(* Logix 5000 project; controller Almacen_2 vendor 1 type 14 code 235 rev 36.11; software revision 36.00 *)

TASK MainTask (continuous, watchdog 500 ms) : MainProgram
TASK SafetyTask (periodic, rate 20 ms, priority 10, watchdog 20 ms) : SafetyProgram

MODULES
   Local : vendor 1 type 14 code 235 (5069 0, rev 36.11)
      EN2TR_Principal : vendor 1 type 12 code 200 (Ethernet 10.12.143.10, rev 10.7, Output RPI 10 ms)
           Point_IO_Conveyor_2:10:O.0   // Spare
           Point_IO_Conveyor_2:10:O.1   // Spare
           Point_IO_Conveyor_2:10:O.2   // Spare
           Point_IO_Conveyor_2:10:O.3   // Spare
           Point_IO_Conveyor_2:10:O.4   // Spare
           Point_IO_Conveyor_2:10:O.5   // Spare
           Point_IO_Conveyor_2:10:O.6   // Spare
           Point_IO_Conveyor_2:10:O.7   // Spare
           Point_IO_Conveyor_2:8:O.5   // Spare
           Point_IO_Conveyor_2:8:O.0   // Reset Válvula General Conveyor 2
           Point_IO_Conveyor_2:8:O.1   // Señal de Impresion de Marcadora Laser
           Point_IO_Conveyor_2:8:O.2   // Lampara indicadora izquierda
           Point_IO_Conveyor_2:8:O.3   // Lampara Cognex 2
           Point_IO_Conveyor_2:8:O.4   // Lampara Cognex 1
           Point_IO_Conveyor_2:8:O.6   // Spare
           Point_IO_Conveyor_2:8:O.7   // Spare
           Point_IO_Almacen_2:1:I.2   // Sensor Piston 1 Horizontal Izquierda
           Point_IO_Almacen_2:1:I.3   // Sensor Piston 1 Horizontal Derecha
           Point_IO_Almacen_2:1:I.4   // Disponible
           Point_IO_Almacen_2:1:I.5   // Sensor Piston 2 Vertical Atras
           Point_IO_Almacen_2:1:I.6   // Sensor Piston 4 Giro Direccion Conveyor
           Point_IO_Almacen_2:1:I.7   // Sensor Piston 4 Giro Direccion Almacen
           Point_IO_Almacen_2:1:I.0   // Disponible
           Point_IO_Almacen_2:1:I.1   // Sensor Piston 3 Griper Arriba
           Point_IO_Conveyor_2:5:I.0   // Sensor Limit Switch Tope
           Point_IO_Conveyor_2:5:I.1   // Sensor Inductivo Entrada desde Almacén (Inicial)
           Point_IO_Conveyor_2:5:I.2   // Robot Fanuc Fence Open
           Point_IO_Conveyor_2:5:I.3   // Robot Fanuc E Stop
           Point_IO_Conveyor_2:5:I.4   // Spare
           Point_IO_Conveyor_2:5:I.5   // Spare
           Point_IO_Conveyor_2:5:I.6   // Spare
           Point_IO_Conveyor_2:5:I.7   // Spare
           Point_IO_Conveyor_2:1:I.0   // Spare
           Point_IO_Conveyor_2:1:I.1   // Spare
           Point_IO_Conveyor_2:1:I.2   // Botón Negro Puerta
           Point_IO_Conveyor_2:1:I.3   // Botón Rojo Puerta
           Point_IO_Conveyor_2:1:I.4   // Contacto Auxiliar Escaner de Seguridad
           Point_IO_Conveyor_2:1:I.5   // Spare
           Point_IO_Conveyor_2:1:I.6   // Sensor Difuso Presencia Lado A Almacen 1-1
           Point_IO_Conveyor_2:1:I.7   // Sensor Difuso Presencia Lado A Almacen 1-2
           Point_IO_Almacen_2:5:O.2   // Disponible
           Point_IO_Almacen_2:5:O.3   // Torreta Roja
           Point_IO_Almacen_2:5:O.0   // Torreta Verde
           Point_IO_Almacen_2:5:O.1   // Torreta Amarilla
           Point_IO_Almacen_2:3:O.1   // Desplazar a Izquierda
           Point_IO_Almacen_2:3:O.2   // Cerrar Gripper
           Point_IO_Almacen_2:3:O.3   // Abrir Gripper
           Point_IO_Almacen_2:3:O.4   // Giro direccion Conveyor
           Point_IO_Almacen_2:3:O.5   // Giro direccion Almacen
           Point_IO_Almacen_2:3:O.6   // Contraer Brazo
           Point_IO_Almacen_2:3:O.7   // Extender Brazo
           Point_IO_Almacen_2:3:O.0   // Desplazar a Derecha
           Point_IO_Conveyor_2:7:O.0   // Piston Horizontal Para Salida de Pieza
           Point_IO_Conveyor_2:7:O.1   // Tope Piston Salida de Producto (freno 8)
           Point_IO_Conveyor_2:7:O.2   // Tope Piston CNC (Freno 5)
           Point_IO_Conveyor_2:7:O.3   // Tope Piston Marcadora Laser (Freno 06)
           Point_IO_Conveyor_2:7:O.4   // Subir Limit Switch
           Point_IO_Conveyor_2:7:O.5   // Tope Piston Cámara Visión
           Point_IO_Conveyor_2:7:O.6   // Piston Cambio de Dirección CNC
           Point_IO_Conveyor_2:7:O.7   // Piston Cambio de Dirección Almacén
           Point_IO_Almacen_2:2:I.0   // Sensor Piston 3 Griper Abajo
           Point_IO_Almacen_2:2:I.2   // Sensor Piston 2 Vertical Adelante
           Point_IO_Almacen_2:2:I.3   // Boton Verde
           Point_IO_Almacen_2:2:I.4   // Dispónible
           Point_IO_Almacen_2:2:I.5   // Disponible
           Point_IO_Almacen_2:2:I.6   // Disponible
           Point_IO_Almacen_2:2:I.1   // Boton Azul
           Point_IO_Almacen_2:2:I.7   // Disponible
           Point_IO_Almacen_2:4:O.0   // Disponible
           Point_IO_Almacen_2:4:O.1   // Dispobible Relevador 1
           Point_IO_Almacen_2:4:O.2   // Disponible Relevador 2
           Point_IO_Almacen_2:4:O.3   // Disponible Relevador 3
           Point_IO_Almacen_2:4:O.4   // Disponible Relevador 4
           Point_IO_Almacen_2:4:O.5   // Disponible Relevador 5
           Point_IO_Almacen_2:4:O.6   // Disponible Relevador 6
           Point_IO_Almacen_2:4:O.7   // Disponible
           Point_IO_Conveyor_2:2:I.0   // Sensor Difuso Presencia Lado B CNC 2-1
           Point_IO_Conveyor_2:2:I.1   // Sensor Difuso Presencia Lado B CNC 2-2
           Point_IO_Conveyor_2:2:I.2   // Sensor Difuso Presencia Lado A CNC 3-1
           Point_IO_Conveyor_2:2:I.3   // Sensor Difuso Presencia Lado A CNC 3-2
           Point_IO_Conveyor_2:2:I.4   // Sensor Inductivo Presente Zona de Marcadora Láser
           Point_IO_Conveyor_2:2:I.5   // Sensor Piston Horizontal Retraido
           Point_IO_Conveyor_2:2:I.6   // Sensor Piston Horizontal Extendido
           Point_IO_Conveyor_2:2:I.7   // Spare
           Point_IO_Conveyor_2:3:I.5   // Sensor Piston Tope Camara Vision
           Point_IO_Conveyor_2:3:I.6   // Cambio de Dirección Extendido Lado B CNC
           Point_IO_Conveyor_2:3:I.7   // Cambio de Dirección Retraido Lado B CNC
           Point_IO_Conveyor_2:3:I.0   // Spare
           Point_IO_Conveyor_2:3:I.1   // Sensor Tope Piston Horizontal (Salida de conveyor)
           Point_IO_Conveyor_2:3:I.2   // Sensor Piston Tope CNC
           Point_IO_Conveyor_2:3:I.3   // Sensor Piston Tope Marcadora Laser
           Point_IO_Conveyor_2:3:I.4   // Límit Switch Arriba
           Point_IO_Conveyor_2:4:I.2   // Sensor Inductivo Izquierdo Almacen
           Point_IO_Conveyor_2:4:I.3   // Sensor Inductivo Posición Lado B CNC
           Point_IO_Conveyor_2:4:I.4   // Spare
           Point_IO_Conveyor_2:4:I.5   // Spare
           Point_IO_Conveyor_2:4:I.6   // Sensor Inductivo Posición Lado A CNC
           Point_IO_Conveyor_2:4:I.7   // Sensor Inductivo Derecho Almacen
           Point_IO_Conveyor_2:4:I.0   // Cambio de Dirección Extendido Lado A Almacén
           Point_IO_Conveyor_2:4:I.1   // Cambio de Dirección Retraido Lado A Almacén
           Point_IO_Conveyor_2:6:I.0   // Spare
           Point_IO_Conveyor_2:6:I.1   // Spare
           Point_IO_Conveyor_2:6:I.2   // Spare
           Point_IO_Conveyor_2:6:I.3   // Spare
           Point_IO_Conveyor_2:6:I.4   // Spare
           Point_IO_Conveyor_2:6:I.5   // Spare
           Point_IO_Conveyor_2:6:I.6   // Spare
           Point_IO_Conveyor_2:6:I.7   // Spare
           Point_IO_Conveyor_2:9:O.0   // Spare
           Point_IO_Conveyor_2:9:O.1   // Spare
           Point_IO_Conveyor_2:9:O.2   // Spare
           Point_IO_Conveyor_2:9:O.3   // Spare
           Point_IO_Conveyor_2:9:O.4   // Spare
           Point_IO_Conveyor_2:9:O.5   // Spare
           Point_IO_Conveyor_2:9:O.6   // Spare
           Point_IO_Conveyor_2:9:O.7   // Spare
         @c7c1ea3c@:Partner : vendor 1 type 14 code 146 (ICP 2, rev 31.11)
         PLC_Principal : vendor 1 type 14 code 148 (ICP 1, rev 31.11, $9b80a274$ RPI 20 ms, $99027f0f$ RPI 20 ms, $04b127b6$ RPI 20 ms, $5697a221$ RPI 20 ms, $7c2d11c0$ RPI 20 ms, $f406f243$ RPI 20 ms, $fc3bde9a$ RPI 20 ms)
      Conveyo_2 : PowerFlex 525-EENET (Ethernet 10.12.143.7, rev 5.1, Output RPI 20 ms)   // Conveyor Derecho
      Cognex_Alm_2 : vendor 678 type 100 code 260 (Ethernet 10.12.143.156, rev 12.2, Output RPI 60 ms)
      Point_IO_Conveyor_2 : 1734-AENTR (Ethernet 10.12.143.43, rev 5.12, Output RPI 20 ms)   // Lado Izquierdo
         E01N023S01 : 1734-IB8 (PointIO 1, rev 3.22)
         E01N023S02 : 1734-IB8 (PointIO 2, rev 3.22)
         E01N023S03 : 1734-IB8 (PointIO 3, rev 3.22)
         E01N023S05 : 1734-IB8 (PointIO 5, rev 3.22)
         E01N023S06 : 1734-IB8 (PointIO 6, rev 3.22)
         E01N023S04 : 1734-IB8 (PointIO 4, rev 3.22)
         E01N023S08 : 1734-OB8 (PointIO 8, rev 3.22)
         E01N023S0 : 1734-OB8 (PointIO 7, rev 3.22)
         E01N023S09 : 1734-OW4 (PointIO 9, rev 3.22)
         E01N023S10 : 1734-OW4 (PointIO 10, rev 3.22)
         E01N023S11 : vendor 1 type 35 code 15 (PointIO 11, rev 2.2, Input RPI 10 ms, Output RPI 20 ms)
              Point_IO_Conveyor_2:11:I.Pt02Data   // E_Stop Coneyor 2 Lierado
              Point_IO_Conveyor_2:11:I.Pt05Data   // Scanner
              Point_IO_Conveyor_2:11:I.Pt01Data   // Spare
              Point_IO_Conveyor_2:11:I.Pt06Data   // Spare
              Point_IO_Conveyor_2:11:I.Pt03Data   // E_Stop Coneyor 2 Presionado
              Point_IO_Conveyor_2:11:I.Pt04Data   // Scanner
              Point_IO_Conveyor_2:11:I.Pt00Data   // Spare
              Point_IO_Conveyor_2:11:I.Pt07Data   // Spare
         E01N023S12 : vendor 1 type 35 code 16 (PointIO 12, rev 2.2, Output RPI 20 ms, Input RPI 10 ms)
              Point_IO_Conveyor_2:12:O.Pt00Data   // S1 PowerFlex Transportador 2
              Point_IO_Conveyor_2:12:O.Pt06Data   // Spare
              Point_IO_Conveyor_2:12:O.Pt05Data   // S2 Robot External E Stop
              Point_IO_Conveyor_2:12:O.Pt02Data   // S1 Robot Fanuc Fence Open
              Point_IO_Conveyor_2:12:O.Pt07Data   // Spare
              Point_IO_Conveyor_2:12:O.Pt01Data   // S2 PowerFlex Transportador 2
              Point_IO_Conveyor_2:12:O.Pt04Data   // S1 Robot External E Stop
              Point_IO_Conveyor_2:12:O.Pt03Data   // S2 Robot Fanuc Fence Open
      Point_IO_Almacen_2 : 1734-AENTR (Ethernet 10.12.143.41, rev 5.12, Output RPI 20 ms)   // Almacen Lado Derecho
         E01N021S01 : 1734-IB8 (PointIO 1, rev 3.22)
         E01N021S02 : 1734-IB8 (PointIO 2, rev 3.22)
         E01N021S03 : 1734-OB8 (PointIO 3, rev 3.22)
         E01N021S04 : 1734-OB8 (PointIO 4, rev 3.22)
         E01N021S05 : 1734-OW4 (PointIO 5, rev 3.22)
         E01N021S06 : vendor 1 type 35 code 15 (PointIO 6, rev 2.2, Input RPI 10 ms, Output RPI 20 ms)
         E01N021S07 : vendor 1 type 35 code 16 (PointIO 7, rev 2.2, Input RPI 10 ms, Output RPI 20 ms)
END_MODULES

TYPE Position_Storage :
STRUCT
   X_Actual : DINT;
   X_Offset : DINT;
   X_Pick : DINT;
   X_Place : DINT;
   X_PlaceOff : DINT;
   Y_Actual : DINT;
   Y_Offset : DINT;
   Y_OffsetMin : DINT;
   Y_OffsetMax : DINT;
   Y_Pick : DINT;
   Y_PickMin : DINT;
   Y_PickMax : DINT;
   Y_Place : DINT;
   Y_PlaceMin : DINT;
   Y_PlaceMax : DINT;
   Y_PlaceOff : DINT;
   Y_PlaceOffMin : DINT;
   Y_PlaceOffMax : DINT;
   Z_Actual : DINT;
   Z_Offset : DINT;
   Z_Pick : DINT;
   Z_Place : DINT;
   Z_PlaceOff : DINT;
   S_Actual : DINT;
   S_Offset : DINT;
   S_Pick : DINT;
   S_Place : DINT;
   S_PlaceOff : DINT;
   SpareBool : BOOL[32];
   spareDint : DINT[10];
   Y_PlaceSafe : DINT;
   Y_PickSafe : DINT;
END_STRUCT
END_TYPE

TYPE Safety :   // TAGS de SAfety para compartir con otro PLC
STRUCT
   Connection_Status : CONNECTION_STATUS;
   DINT : DINT;
END_STRUCT
END_TYPE

ADD_ON_INSTRUCTION Debounce   (* revision 1.0, vendor Premier Tech Ltd, ExecuteEnableInFalse *)
// Revision note:
// 1.0 Master 1st release
VAR_INPUT
   FilterOnTimerPreset : ALIAS FOR FilterOnTimer.PRE; {required}   // Digital input filter time preset (ON)
   FilterOffTimerPreset : ALIAS FOR FilterOffTimer.PRE; {required}   // Digital input filter time preset (OFF)
END_VAR
VAR_OUTPUT
   B : BOOL; {access Read Only, visible}   // Digital input filtered signal
   BFT : BOOL; {access Read Only}   // Falling transient: digital input filtered signal
   BRT : BOOL; {access Read Only}   // Rising transient: digital input filtered signal
   I : BOOL; {access Read Only}   // Digital input raw signal
   IFT : BOOL; {access Read Only}   // Falling transient: digital input raw signal
   IRT : BOOL; {access Read Only}   // Rising transient: digital input raw signal
END_VAR
VAR
   FilterOffTimer : TIMER := (PRE := 50);   // Digital input filter time (OFF)
   FilterOnTimer : TIMER := (PRE := 50);   // Digital input filter time (ON)
   B_Osr : BOOL; {access None}
   B_Osf : BOOL; {access None}
   I_Osr : BOOL; {access None}
   I_Osf : BOOL; {access None}
END_VAR

ROUTINE EnableInFalse   (* ladder *)
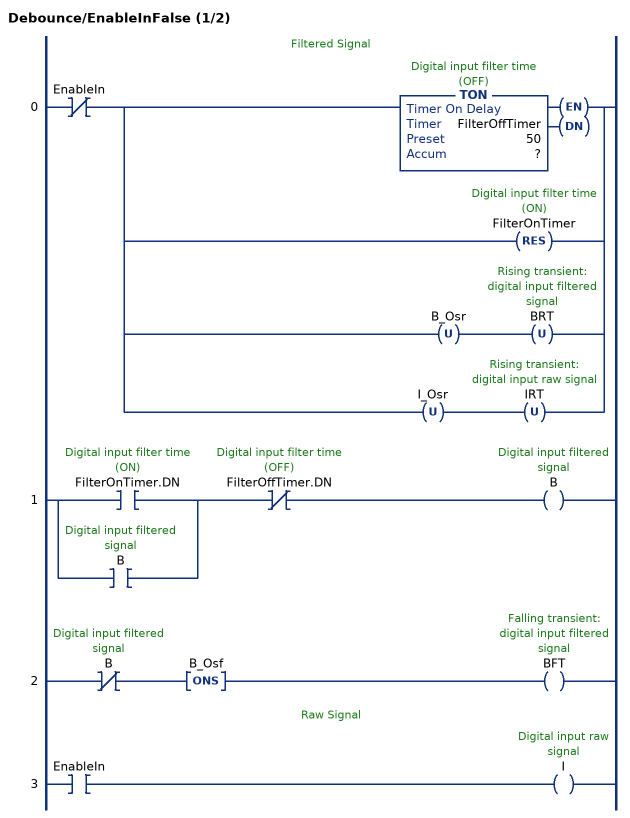
   // Filtered Signal
   0: XIO(EnableIn)[TON(FilterOffTimer,?,?) ,RES(FilterOnTimer) ,OTU(B_Osr) OTU(BRT) ,OTU(I_Osr) OTU(IRT) ];
   1: [XIC(FilterOnTimer.DN) ,XIC(B) ]XIO(FilterOffTimer.DN)OTE(B);
   2: XIO(B)ONS(B_Osf)OTE(BFT);
   // Raw Signal
   3: XIC(EnableIn)OTE(I);
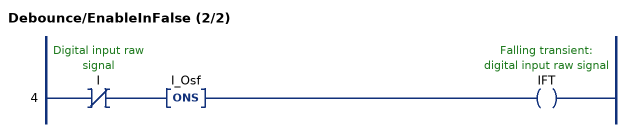
   4: XIO(I)ONS(I_Osf)OTE(IFT);
END_ROUTINE

ROUTINE Logic   (* ladder *)
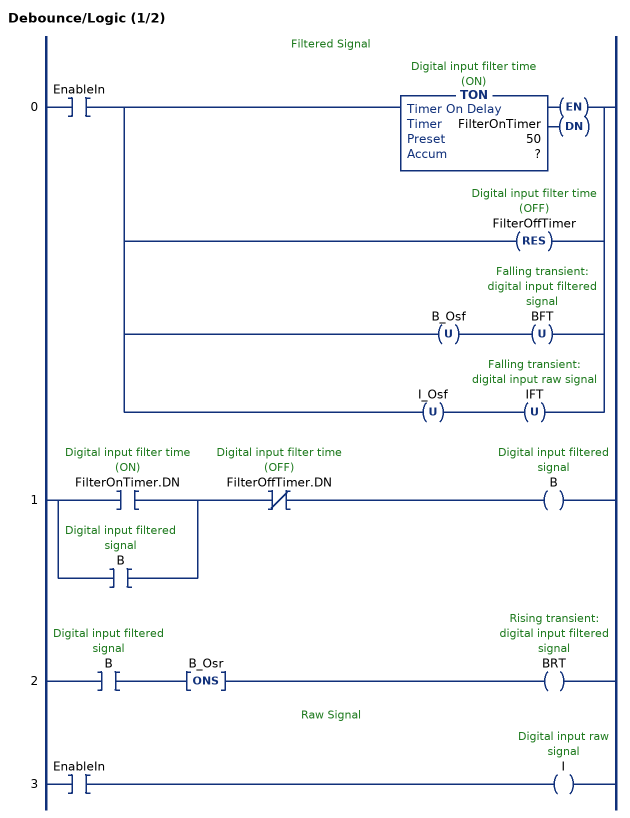
   // Filtered Signal
   0: XIC(EnableIn)[TON(FilterOnTimer,?,?) ,RES(FilterOffTimer) ,OTU(B_Osf) OTU(BFT) ,OTU(I_Osf) OTU(IFT) ];
   1: [XIC(FilterOnTimer.DN) ,XIC(B) ]XIO(FilterOffTimer.DN)OTE(B);
   2: XIC(B)ONS(B_Osr)OTE(BRT);
   // Raw Signal
   3: XIC(EnableIn)OTE(I);
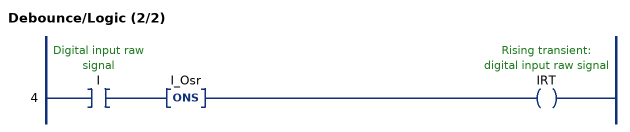
   4: XIC(I)ONS(I_Osr)OTE(IRT);
END_ROUTINE
END_ADD_ON_INSTRUCTION

VAR_GLOBAL   (* controller tags *)
   Abrir_Gripper : BOOL;
   Abrir_Gripper_01 : BOOL;
   Alarms_OK : BOOL := 1;
   Alm2_Home : BOOL := 1;
   Alm2_S2 : BOOL;
   Alm2_X2 : BOOL;
   AlmPosReq : DINT;
   At_Pos_Alm_2 : DINT;
   Auto_Conv_2 : BOOL := 1;
   Auto_Enabled : BOOL := 1;
   B_Reset_Posicion_kinetix : DINT := 1; {produced}
   BACK_SQUADRA_1 : TIMER := (PRE := 6000);
   BACK_SQUADRA_2 : TIMER := (PRE := 8000);
   Bit_CambioDir_Conv_2 : BOOL;
   Bit_CambioDirAlm_Conv_2 : BOOL;
   Bit_FinDeCarreraConv_2 : BOOL;
   Bit_Pruebas : DINT := -2147483520;
   Bit_Reset_ValvulaGeneral_Conv_2 : BOOL := 1;
   BK_SQUA_2 : BOOL;
   Btn_Negro_Conv_2 : BOOL;   // Botón Negro Puerta de Conveyor 2
   Btn_Rojo_Conv_2 : BOOL;   // Botón Rojo Puerta de Conveyor 2
   CambioDir_Ext_Almacen_Conv_1 : BOOL;   // Sensor Cambio de Dirección Extendido Lado A (Almacén)
   CambioDir_Ext_Almacen_Conv_2 : BOOL;   // Sensor Cambio de Dirección Extendido Lado A Almacén
   CambioDir_Ext_CNC_Conv_1 : BOOL;   // Sensor Cambio de Dirección Extendido Lado B (CNC)
   CambioDir_Ext_CNC_Conv_2 : BOOL;   // Cambio de Dirección Extendido Lado B CNC
   CambioDir_Ret_Almacen_Conv_1 : BOOL := 1;   // Sensor Cambio de Dirección Retraido Lado A (Almacén)
   CambioDir_Ret_Almacen_Conv_2 : BOOL := 1;   // Sensor Cambio de Dirección Retraido Lado A Almacén
   CambioDir_Ret_CNC_Conv_1 : BOOL;   // Sensor Cambio de Dirección Retraido Lado B (CNC)
   CambioDir_Ret_CNC_Conv_2 : BOOL := 1;   // Cambio de Dirección Retraido Lado B CNC
   CellAuto : BOOL := 1;
   cerrar_gripper : BOOL;
   CERRAr_gripper_01 : BOOL;
   Cmd_CloseGripper : BOOL;
   Cmd_OpenGripper : BOOL;
   Cmd_ServoHome : BOOL;
   Cmd_StoS1Pos : BOOL;   // Giro Lado de Almacén 2
   Cmd_StoS2Pos : BOOL;   // Giro Lado de Conveyor 2
   Cmd_XtoX1Pos : BOOL;   // Lado Entrada almacén 2
   Cmd_XtoX2Pos : BOOL;   // Lado Salida Almacén 2
   Cmd_YPickSafe : BOOL;
   Cmd_YPlaceSAfe : BOOL;
   Cmd_YSafePos : BOOL;
   Cmd_YtoYOff : BOOL;
   Cmd_YtoYPick : BOOL;
   Cmd_YtoYPlace : BOOL;
   Cmd_YtoYPlaceOffset : BOOL;
   Cmd_ZtoZ1Pos : BOOL;   // Lado del Conveyor 2
   Cmd_ZtoZ2Pos : BOOL;   // Lado del Almacén 2
   CON_OFF_STOP_2 : TIMER := (PRE := 5000);
   CONT_PASOS : COUNTER := (PRE := 13);
   Continuar_Secuencia_en_Conveyor_1 : BOOL;   // Bit de Terminación de Procesos de CNC 1 y Mesa KUKA
   Continuar_Secuencia_en_Conveyor_2 : BOOL;
   Conv_2_Actual_Step : DINT := 50;
   Conv_2_Aux : INT := 1;
   Conv_2_Perm_OnDly : TIMER[32] := ([0].PRE := 100, [1].PRE := 100, [2].PRE := 100, [3].PRE := 100, [4].PRE := 500, [5].PRE := 250, [6].PRE := 100, [7].PRE := 100, [8].PRE := 100, [9].PRE := 100, [10].PRE := 1000, [11].PRE := 20000, [12].PRE := 100, [13].PRE := 100, [14].PRE := 100, [15].PRE := 100, [16].PRE := 100, [17].PRE := 100, [18].PRE := 100, [19].PRE := 100, [20].PRE := 100, [21].PRE := 100);
   Conv_2_Step : DINT := 32;
        .0   // ESPERA SEÑAL DE INICIO Y VERIFICA QUE EL TRANSPORTADOR SE ENCUENTRE VACÍO
        .10   // ESPERA 1 SEGUNDO CON EL PISTÓN TOPE ARRIBA Y DETIENE EL TRANSPORTADOR
        .14   // ESPERA QUE SENSORES DEJEN DE VER PIEZA EN FIN DE TRANSPORTADOR
        .3   // AVANZA HASTA DEJAR DE VER LA PIEZA EN LOS SENSORES DEL ÁREA DE CNC
        .17   // ELEVA TOPE DE PISTÓN Y ESPERA CONFIRMACIÓN DE GRIPPER EN POSICIÓN
        .8   // ESPERA DETECTAR PIEZA EN AREA DE MARCADORA LÁSER
        .19   // RETORNA PISTÓN.
        .9   // ESPERA QUE PIEZA AVANCE A ZONA DE MARCADORA LÁSER
        .5   // ESPERA A QUE EL ROBOT FANUC CONFIRME PIEZA DEVUELTA EN EL TRANSPORTADOR
        .2   // ESPERA LLEGADA DE PIEZA A FIN DE TRANSPORTADOR
        .1   // CONFIRMA NUEVA PIEZA EN TRANSPORTADOR
        .11   // TIEMPO DE TRABAJO DE MARCADORA LÁSER
        .12   // BAJA PISTÓN Y ESPERA CONFIRMACIÓN
        .20   // BAJA TOPE DE PISTÓN
        .21   // ESPERA CONFIRMACIÓN DE PIEZA RETIRADA
        .4   // VERIFICA QUE LA PUERTA DEL CNC ESTÉ ABIERTA
        .13   // ESPERA A QUE PIEZA LLEGUE AL SENSOR DE FIN DE TRANSPORTADOR
        .6   // MUEVE LA PIEZA PARA RETORNO AL ALMACÉN.
        .7   // ESPERA PISTÓN RETRAÍDO
        .15   // EXTIENDE PISTÓN Y ESPERA CONFIRMACIÓN
        .16   // ESPERA PISTÓN RETRAÍDO
        .18   // EXTIENDE PISTÓN PARA MOVER PIEZA HACIA GRIPPER
   Conv_2_Vacio_Inicial : BOOL := 1;
   Ctrl_Kinetix_A2 : DINT := 1; {produced}   // Habilitar Kinetix
   Cycle_Start : BOOL;
   Debounce_Alimentacion_Conv_2 : Debounce := (FilterOffTimerPreset := 3000);
   Debounce_Almacen_Conv_1 : Debounce := (FilterOffTimerPreset := 3000);
   Debounce_Almacen_Conv_2 : Debounce := (FilterOffTimerPreset := 3000);
   Debounce_CNC_2_Conv_1 : Debounce := (FilterOffTimerPreset := 3000);
   Debounce_CNC_2_Conv_2 : Debounce := (FilterOffTimerPreset := 3000);
   Debounce_CNC_Conv_2 : Debounce := (FilterOffTimerPreset := 3000);
   Debounce_Entrada_Conv_2 : Debounce := (FilterOffTimerPreset := 3000);
   Debounce_Marcadora_Conv_1 : Debounce := (FilterOffTimerPreset := 100);
   Debounce_Marcadora_Conv_2 : Debounce := (FilterOffTimerPreset := 100);
   Dir_Almacen_01 : BOOL;
   Dir_Almacen_2 : BOOL;
   DIR_CONV_01 : BOOL;
   Dir_Conveyor : BOOL;
   Done_Kinetx : DINT;
   Done_Kinetx_ok : BOOL;
   Done_Kinetx_ok_01 : BOOL;
   Done_Step_00_Conv_1 : BOOL;
   Done_Step_00_Conv_2 : BOOL;
   Done_Step_01_Conv_1 : BOOL;
   Done_Step_01_Conv_2 : BOOL;
   Done_Step_02_Conv_1 : BOOL;
   Done_Step_02_Conv_2 : BOOL;
   Done_Step_03_Conv_1 : BOOL;
   Done_Step_03_Conv_2 : BOOL;
   Done_Step_04_Conv_1 : BOOL;
   Done_Step_04_Conv_2 : BOOL;
   Done_Step_05_Conv_1 : BOOL;
   Done_Step_05_Conv_2 : BOOL;
   Done_Step_06_Conv_1 : BOOL;
   Done_Step_06_Conv_2 : BOOL;
   Done_Step_07_Conv_1 : BOOL;
   Done_Step_07_Conv_2 : BOOL;
   Done_Step_08_Conv_1 : BOOL;
   Done_Step_08_Conv_2 : BOOL;
   Done_Step_09_Conv_1 : BOOL;
   Done_Step_09_Conv_2 : BOOL;
   Done_Step_10_Conv_1 : BOOL;
   Done_Step_10_Conv_2 : BOOL;
   Done_Step_11_Conv_1 : BOOL;
   Done_Step_11_Conv_2 : BOOL;
   Done_Step_12_Conv_1 : BOOL;
   Done_Step_12_Conv_2 : BOOL;
   Done_Step_13_Conv_1 : BOOL;
   Done_Step_13_Conv_2 : BOOL;
   Done_Step_14_Conv_1 : BOOL;
   Done_Step_14_Conv_2 : BOOL;
   Done_Step_15_Conv_1 : BOOL;
   Done_Step_15_Conv_2 : BOOL;
   Done_Step_16_Conv_1 : BOOL;
   Done_Step_16_Conv_2 : BOOL;
   Done_Step_17_Conv_1 : BOOL;
   Done_Step_17_Conv_2 : BOOL;
   Done_Step_18_Conv_1 : BOOL;
   Done_Step_18_Conv_2 : BOOL;
   Done_Step_19_Conv_1 : BOOL;
   Done_Step_19_Conv_2 : BOOL;
   Done_Step_20_Conv_1 : BOOL;
   Done_Step_20_Conv_2 : BOOL;
   Done_Step_21_Conv_1 : BOOL;
   Done_Step_21_Conv_2 : BOOL;
   Done_Step_22_Conv_1 : BOOL;
   Done_Step_23_Conv_1 : BOOL;
   Done_Step_24_Conv_1 : BOOL;
   Done_Step_25_Conv_1 : BOOL;
   Done_Step_26_Conv_1 : BOOL;
   Done_Step_27_Conv_1 : BOOL;
   Done_Step_28_Conv_1 : BOOL;
   Done_Step_29_Conv_1 : BOOL;
   Done_Step_30_Conv_1 : BOOL;
   Done_Step_31_Conv_1 : BOOL;
   Done_Step_32_Conv_1 : BOOL;
   Done_Step_33_Conv_1 : BOOL;
   Done_Step_34_Conv_1 : BOOL;
   Done_Step_35_Conv_1 : BOOL;
   Done_Step_36_Conv_1 : BOOL;
   Done_Step_37_Conv_1 : BOOL;
   Done_Step_38_Conv_1 : BOOL;
   Done_Step_39_Conv_1 : BOOL;
   Done_Step_40_Conv_1 : BOOL;
   E4_timer1 : TIMER := (PRE := 1500);
   enclave_paso22 : BOOL;
   End_Alm_2_Start_Conv_2 : BOOL;
   End_Alm_Start_Conv : BOOL;   // Almacén Entrega Pieza a Conveyor
   End_Conv_Start_Alm : BOOL;
   End_Conv_Start_Alm_2 : BOOL;
   Entrada_Almacen : BOOL;
   equuipo_en_pos : BOOL;
   equuipo_en_pos_entrada : BOOL;
   Espe_Pos_6 : BOOL;
   Espera_Cerrar_Griper : TIMER := (PRE := 1500);
   Espera_Plato : BOOL;
   Estops_Ok : BOOL := 1;
   EStops_OK_External_A1 : DINT := 3;
   ETAPA_FIN : BOOL;
   Fanuc_CNC_Bypass : BOOL;
   Fanuc_Griper_Cerrado_Conv_1 : BOOL := 1;   // Señal desde Robot Fanuc Para indicar el Cerrado de Griper Exclusivo Conveyor 1
   Fanuc_Posicion_Dejar_Pieza_Mesa_1 : BOOL := 1;   // Señal de Posición del Robot Fanuc para dejar Pieza en Pistón 1 de la Mesa Kuka Conveyor 1
   Fanuc_Posicion_Segura_CNC_1 : BOOL := 1;   // Posición Segura de Robot Fanuc Después de Dejar Pieza en CNC 1 Conveyor 1
   Fanuc_Posicion_Segura_Mesa_1 : BOOL := 1;   // Posición Segura Frente a Mesa Kuka Conveyor 1
   Fanuc_RetornoPieza_Conv_2 : BOOL;
   FINAL_RESET : BOOL;
   Fixture_Sensor_Direccion_Conveyor_2 : BOOL;
   Freq_cnv1 : DINT := 5000;
   FromConv_PieceDone : BOOL;
   FromRobot_Confirm : BOOL;
   Green_Light_Alm_2 : BOOL;
   HMI_Conveyor_Reset_Sequence : BOOL;
   HMI_Conveyor_Select_Sequence : BOOL;
   HMI_Conveyor_Start : BOOL;
   HMI_Start : BOOL;
   Home_Wh_Dn : BOOL;
   Home_Wh_Req : BOOL;
   HomeDone : BOOL;
   HomeRequired : BOOL;
   HomeStep0 : BOOL := 1;   // Request for Home
   HomeStep1 : BOOL;   // Evaluar Condiones a seguir
   HomeStep10 : BOOL;
   HomeStep11 : BOOL;
   HomeStep2 : BOOL;   // S to S1
   HomeStep3 : BOOL;   // S to S2
   HomeStep4 : BOOL;   // Y to Y Home
   HomeStep5 : BOOL;   // Z to Z1
   HomeStep6 : BOOL;   // S to S1
   HomeStep7 : BOOL;   // X to X1
   HomeStep8 : BOOL;   // Open Gripper
   Homestep9 : BOOL;   // Homed
   HomeStoSeqToTec81 : DINT; {produced}
   Homming : BOOL;
   Homming_Wh2 : BOOL;
   Homming_Wh2_Cycle : BOOL;
   In_Pos_Alm_2 : DINT;
   IndexPickStorage1 : DINT;
   IndexPickStorage2 : DINT := 1;
   IndexPlaceStorage1 : DINT;
   IndexPlaceStorage2 : DINT;
   InicioCiclo : BOOL;
   Interlocks_Ok : BOOL := 1;
   Kinetix_Pos : DINT; {produced}
   Kinetix_Running : BOOL;
   KUKA_Posicion_Segura : BOOL := 1;   // Posición Segura del Robot KUKA Sin Movimiento, en Espera de Recibir Pieza
   KUKA_Proceso_Terminado_Conv_1 : BOOL;   // Proceso Terminado para Pieza de Conveyor 1
   LigthCurtain2_Ok : BOOL := 1;
   Limit_UP_Conv_2 : BOOL;   // Subir Limit Switch Conveyor 2
   Load : BOOL;
   M0 : BOOL;
   M1 : BOOL;
   m100 : DINT;
   M11 : BOOL := 1;
   M2 : BOOL;
   M3 : BOOL;
   M4 : BOOL;
   M5 : BOOL;
   M6 : BOOL;
   M66 : BOOL;
   M7 : BOOL;
   M77 : BOOL;
   M8 : BOOL;
   M_DOWN_STOPER_1 : BOOL;
   Manual_Conv_2 : BOOL;
   Marcadora_Print : BOOL;   // Señal para la Marcadora de imprimir
   Mesa_Kuka_Piston_1_Abierto : BOOL := 1;   // Pistón Para Sujetar Pieza de conveyor 1 Abierta Conveyor 1
   Mover_piston : BOOL;
   ok_com : BOOL;
   ONS_Marcadora : BOOL;
   Operacion_Salida : BOOL;
   P2_Adelante : BOOL;
   Paso_11 : BOOL;
   Paso_1_OK : BOOL := 1;
   PASO_L1 : BOOL;
   PASO_L2 : BOOL;
   PASO_NUM : DINT := 1073741824;
   PB_ARRANQUE_SISTEMA : BOOL;
   PB_PARO_SISTEMA : BOOL;
   Permissive_HomeStep0 : BOOL;
   Permissive_homeStep1 : BOOL;
   Permissive_HomeStep10 : BOOL;
   Permissive_HomeStep11 : BOOL;
   Permissive_HomeStep2 : BOOL;
   Permissive_HomeStep3 : BOOL;
   Permissive_HomeStep4 : BOOL;
   Permissive_HomeStep5 : BOOL;
   Permissive_HomeStep6 : BOOL;
   Permissive_HomeStep7 : BOOL;
   Permissive_HomeStep8 : BOOL;
   Permissive_HomeStep9 : BOOL;
   Permissive_Step0 : BOOL;
   Permissive_Step1 : BOOL;
   Permissive_Step10 : BOOL;
   Permissive_Step11 : BOOL;
   Permissive_Step12 : BOOL;
   Permissive_Step13 : BOOL;
   Permissive_Step14 : BOOL;
   Permissive_Step15 : BOOL;
   Permissive_Step16 : BOOL;
   Permissive_Step17 : BOOL;
   Permissive_Step18 : BOOL;
   Permissive_Step19 : BOOL;
   Permissive_Step2 : BOOL;
   Permissive_Step20 : BOOL;
   Permissive_Step21 : BOOL;
   Permissive_Step22 : BOOL;
   Permissive_Step23 : BOOL;
   Permissive_Step24 : BOOL;
   Permissive_Step25 : BOOL;
   Permissive_Step26 : BOOL;
   Permissive_Step27 : BOOL;
   Permissive_Step3 : BOOL;
   Permissive_Step4 : BOOL;
   Permissive_Step5 : BOOL;
   Permissive_Step6 : BOOL;
   Permissive_Step7 : BOOL;
   Permissive_Step8 : BOOL;
   Permissive_Step9 : BOOL;
   PF_On_525_Conv_2 : BOOL;   // Encender/Apagar PowerFlex Conveyor 2
   PickPosition : Position_Storage := (X_Offset := 2, X_Pick := 1, X_Place := 1, X_PlaceOff := 2, Y_Offset := 910, Y_OffsetMin := 909, Y_OffsetMax := 911, Y_Pick := 900, Y_PickMin := 899, Y_PickMax := 901, Y_Place := 345, Y_PlaceMin := 344, Y_PlaceMax := 346, Y_PlaceOff := 500, Y_PlaceOffMin := 364, Y_PlaceOffMax := 366, Z_Offset := 1, Z_Pick := 2, Z_Place := 2, Z_PlaceOff := 1, S_Offset := 2, S_Pick := 1, S_Place := 1, S_PlaceOff := 2, Y_PlaceSafe := 345, Y_PickSafe := 900);
   PickPositionPorduced : Position_Storage;
   PickPositionProd : Position_Storage := (X_Offset := 2, X_Pick := 1, X_Place := 1, X_PlaceOff := 2, Y_Offset := 910, Y_OffsetMin := 909, Y_OffsetMax := 911, Y_Pick := 900, Y_PickMin := 899, Y_PickMax := 901, Y_Place := 345, Y_PlaceMin := 344, Y_PlaceMax := 346, Y_PlaceOff := 500, Y_PlaceOffMin := 364, Y_PlaceOffMax := 366, Z_Offset := 1, Z_Pick := 2, Z_Place := 2, Z_PlaceOff := 1, S_Offset := 2, S_Pick := 1, S_Place := 1, S_PlaceOff := 2, Y_PlaceSafe := 345, Y_PickSafe := 900); {produced}
   Pist_Hor_Der_A2 : BOOL;
   Pist_Hor_Izq_A2 : BOOL;   // Mover piston 1 Horizontal izquierda
   Piston_Adelante : INT;
   Piston_Adelante_0 : BOOL;
   piston_atras : INT;
   Piston_CambioDir_Almacen_Conv_2 : BOOL;   // Cambiar Direccion de Pieza Lado Almacen Conveyor 2
   Piston_CambioDir_CNC_Conv_2 : BOOL;   // Cambiar Dirección de Pieza Lado CNC Conveyor 2
   Piston_Horizontal_Conv_2 : BOOL := 1;   // Extender Pistón Horizontal del Conveyor 2
   Piston_vertical_salida : BOOL;
   PlacePosition : Position_Storage;
   PlacesStorage1 : Position_Storage[20] := ([1].X_Offset := 2, [1].X_Pick := 1, [1].X_Place := 1, [1].X_PlaceOff := 2, [1].Z_Offset := 1, [1].Z_Pick := 2, [1].Z_Place := 2, [1].Z_PlaceOff := 1, [1].S_Offset := 2, [1].S_Pick := 1, [1].S_Place := 1, [1].S_PlaceOff := 2, [2].X_Offset := 2, [2].X_Pick := 1, [2].X_Place := 1, [2].X_PlaceOff := 2, [2].Z_Offset := 1, [2].Z_Pick := 2, [2].Z_Place := 2, [2].Z_PlaceOff := 1, [2].S_Offset := 2, [2].S_Pick := 1, [2].S_Place := 1, [2].S_PlaceOff := 2, [3].X_Offset := 2, [3].X_Pick := 1, [3].X_Place := 1, [3].X_PlaceOff := 2, [3].Z_Offset := 1, [3].Z_Pick := 2, [3].Z_Place := 2, [3].Z_PlaceOff := 1, [3].S_Offset := 2, [3].S_Pick := 1, [3].S_Place := 1, [3].S_PlaceOff := 2, [4].X_Offset := 2, [4].X_Pick := 1, [4].X_Place := 1, [4].X_PlaceOff := 2, [4].Z_Offset := 1, [4].Z_Pick := 2, [4].Z_Place := 2, [4].Z_PlaceOff := 1, [4].S_Offset := 2, [4].S_Pick := 1, [4].S_Place := 1, [4].S_PlaceOff := 2, [5].X_Offset := 2, [5].X_Pick := 1, [5].X_Place := 1, [5].X_PlaceOff := 2, [5].Z_Offset := 1, [5].Z_Pick := 2, [5].Z_Place := 2, [5].Z_PlaceOff := 1, [5].S_Offset := 2, [5].S_Pick := 1, [5].S_Place := 1, [5].S_PlaceOff := 2,
        [6].X_Offset := 2, [6].X_Pick := 1, [6].X_Place := 1, [6].X_PlaceOff := 2, [6].Z_Offset := 1, [6].Z_Pick := 2, [6].Z_Place := 2, [6].Z_PlaceOff := 1, [6].S_Offset := 2, [6].S_Pick := 1, [6].S_Place := 1, [6].S_PlaceOff := 2, [7].X_Offset := 1, [7].X_Pick := 2, [7].X_Place := 2, [7].X_PlaceOff := 1, [7].Z_Offset := 1, [7].Z_Pick := 2, [7].Z_Place := 2, [7].Z_PlaceOff := 1, [7].S_Offset := 2, [7].S_Pick := 1, [7].S_Place := 1, [7].S_PlaceOff := 2, [8].X_Offset := 1, [8].X_Pick := 2, [8].X_Place := 2, [8].X_PlaceOff := 1, [8].Z_Offset := 1, [8].Z_Pick := 2, [8].Z_Place := 2, [8].Z_PlaceOff := 1, [8].S_Offset := 2, [8].S_Pick := 1, [8].S_Place := 1, [8].S_PlaceOff := 2, [9].X_Offset := 1, [9].X_Pick := 2, [9].X_Place := 2, [9].X_PlaceOff := 1, [9].Z_Offset := 1, [9].Z_Pick := 2, [9].Z_Place := 2, [9].Z_PlaceOff := 1, [9].S_Offset := 2, [9].S_Pick := 1, [9].S_Place := 1, [9].S_PlaceOff := 2, [10].X_Offset := 1, [10].X_Pick := 2, [10].X_Place := 2, [10].X_PlaceOff := 1, [10].Z_Offset := 1, [10].Z_Pick := 2, [10].Z_Place := 2, [10].Z_PlaceOff := 1, [10].S_Offset := 2, [10].S_Pick := 1, [10].S_Place := 1, [10].S_PlaceOff := 2,
        [11].X_Offset := 1, [11].X_Pick := 2, [11].X_Place := 2, [11].X_PlaceOff := 1, [11].Z_Offset := 1, [11].Z_Pick := 2, [11].Z_Place := 2, [11].Z_PlaceOff := 1, [11].S_Offset := 2, [11].S_Pick := 1, [11].S_Place := 1, [11].S_PlaceOff := 2, [12].X_Offset := 1, [12].X_Pick := 2, [12].X_Place := 2, [12].X_PlaceOff := 1, [12].Z_Offset := 1, [12].Z_Pick := 2, [12].Z_Place := 2, [12].Z_PlaceOff := 1, [12].S_Offset := 2, [12].S_Pick := 1, [12].S_Place := 1, [12].S_PlaceOff := 2, [13].X_Offset := 2, [13].X_Pick := 1, [13].X_Place := 1, [13].X_PlaceOff := 2, [13].Z_Offset := 2, [13].Z_Pick := 1, [13].Z_Place := 1, [13].Z_PlaceOff := 2, [13].S_Actual := 1, [13].S_Offset := 2, [13].S_Pick := 2, [13].S_Place := 1);
   PlacesStorage2 : Position_Storage[20] := ([1].X_Offset := 2, [1].X_Pick := 1, [1].X_Place := 1, [1].X_PlaceOff := 2, [1].Y_Offset := 910, [1].Y_OffsetMin := 909, [1].Y_OffsetMax := 911, [1].Y_Pick := 900, [1].Y_PickMin := 899, [1].Y_PickMax := 901, [1].Y_Place := 345, [1].Y_PlaceMin := 344, [1].Y_PlaceMax := 346, [1].Y_PlaceOff := 500, [1].Y_PlaceOffMin := 364, [1].Y_PlaceOffMax := 366, [1].Z_Offset := 1, [1].Z_Pick := 2, [1].Z_Place := 2, [1].Z_PlaceOff := 1, [1].S_Offset := 2, [1].S_Pick := 1, [1].S_Place := 1, [1].S_PlaceOff := 2, [1].Y_PlaceSafe := 345, [1].Y_PickSafe := 900, [2].X_Offset := 2, [2].X_Pick := 1, [2].X_Place := 1, [2].X_PlaceOff := 2, [2].Y_Offset := 732, [2].Y_Pick := 722, [2].Y_Place := 345, [2].Y_PlaceOff := 500, [2].Z_Offset := 1, [2].Z_Pick := 2, [2].Z_Place := 2, [2].Z_PlaceOff := 1, [2].S_Offset := 2, [2].S_Pick := 1, [2].S_Place := 1, [2].S_PlaceOff := 2, [2].Y_PlaceSafe := 345, [2].Y_PickSafe := 722, [3].X_Offset := 2, [3].X_Pick := 1, [3].X_Place := 1, [3].X_PlaceOff := 2, [3].Y_Offset := 553, [3].Y_Pick := 543, [3].Y_Place := 345, [3].Y_PlaceOff := 500, [3].Z_Offset := 1, [3].Z_Pick := 2, [3].Z_Place := 2, [3].Z_PlaceOff := 1, [3].S_Offset := 2, [3].S_Pick := 1, [3].S_Place := 1, [3].S_PlaceOff := 2,
        [3].Y_PlaceSafe := 345, [3].Y_PickSafe := 543, [4].X_Offset := 2, [4].X_Pick := 1, [4].X_Place := 1, [4].X_PlaceOff := 2, [4].Y_Offset := 376, [4].Y_Pick := 366, [4].Y_Place := 345, [4].Y_PlaceOff := 500, [4].Z_Offset := 1, [4].Z_Pick := 2, [4].Z_Place := 2, [4].Z_PlaceOff := 1, [4].S_Offset := 2, [4].S_Pick := 1, [4].S_Place := 1, [4].S_PlaceOff := 2, [4].Y_PlaceSafe := 345, [4].Y_PickSafe := 366, [5].X_Offset := 2, [5].X_Pick := 1, [5].X_Place := 1, [5].X_PlaceOff := 2, [5].Y_Offset := 199, [5].Y_Pick := 189, [5].Y_Place := 345, [5].Y_PlaceOff := 500, [5].Z_Offset := 1, [5].Z_Pick := 2, [5].Z_Place := 2, [5].Z_PlaceOff := 1, [5].S_Offset := 2, [5].S_Pick := 1, [5].S_Place := 1, [5].S_PlaceOff := 2, [5].Y_PlaceSafe := 345, [5].Y_PickSafe := 189, [6].X_Offset := 2, [6].X_Pick := 1, [6].X_Place := 1, [6].X_PlaceOff := 2, [6].Y_Offset := 20, [6].Y_Pick := 10, [6].Y_Place := 345, [6].Y_PlaceOff := 500, [6].Z_Offset := 1, [6].Z_Pick := 2, [6].Z_Place := 2, [6].Z_PlaceOff := 1, [6].S_Offset := 2, [6].S_Pick := 1, [6].S_Place := 1, [6].S_PlaceOff := 2, [6].Y_PlaceSafe := 345, [6].Y_PickSafe := 10, [7].X_Offset := 1, [7].X_Pick := 2, [7].X_Place := 2, [7].X_PlaceOff := 1,
        [7].Z_Offset := 1, [7].Z_Pick := 2, [7].Z_Place := 2, [7].Z_PlaceOff := 1, [7].S_Offset := 2, [7].S_Pick := 1, [7].S_Place := 1, [7].S_PlaceOff := 2, [8].X_Offset := 1, [8].X_Pick := 2, [8].X_Place := 2, [8].X_PlaceOff := 1, [8].Z_Offset := 1, [8].Z_Pick := 2, [8].Z_Place := 2, [8].Z_PlaceOff := 1, [8].S_Offset := 2, [8].S_Pick := 1, [8].S_Place := 1, [8].S_PlaceOff := 2, [9].X_Offset := 1, [9].X_Pick := 2, [9].X_Place := 2, [9].X_PlaceOff := 1, [9].Z_Offset := 1, [9].Z_Pick := 2, [9].Z_Place := 2, [9].Z_PlaceOff := 1, [9].S_Offset := 2, [9].S_Pick := 1, [9].S_Place := 1, [9].S_PlaceOff := 2, [10].X_Offset := 1, [10].X_Pick := 2, [10].X_Place := 2, [10].X_PlaceOff := 1, [10].Z_Offset := 1, [10].Z_Pick := 2, [10].Z_Place := 2, [10].Z_PlaceOff := 1, [10].S_Offset := 2, [10].S_Pick := 1, [10].S_Place := 1, [10].S_PlaceOff := 2, [11].X_Offset := 1, [11].X_Pick := 2, [11].X_Place := 2, [11].X_PlaceOff := 1, [11].Z_Offset := 1, [11].Z_Pick := 2, [11].Z_Place := 2, [11].Z_PlaceOff := 1, [11].S_Offset := 2, [11].S_Pick := 1, [11].S_Place := 1, [11].S_PlaceOff := 2, [12].X_Offset := 1, [12].X_Pick := 2, [12].X_Place := 2, [12].X_PlaceOff := 1,
        [12].Z_Offset := 1, [12].Z_Pick := 2, [12].Z_Place := 2, [12].Z_PlaceOff := 1, [12].S_Offset := 2, [12].S_Pick := 1, [12].S_Place := 1, [12].S_PlaceOff := 2, [13].X_Offset := 2, [13].X_Pick := 1, [13].X_Place := 1, [13].X_PlaceOff := 2, [13].Z_Offset := 2, [13].Z_Pick := 1, [13].Z_Place := 1, [13].Z_PlaceOff := 2, [13].S_Actual := 1, [13].S_Offset := 2, [13].S_Pick := 2, [13].S_Place := 1);
   PLATO_POS : BOOL;
   plato_salida : BOOL;
   Pos_00_Almacen_2 : BOOL;
   Pos_00_Amacen_2 : BOOL;
   POS_00_Kinetix : BOOL;
   POS_00_Kinetix_01 : BOOL;
   Pos_01_Almacen_2 : BOOL;
   POS_01_Kinetix : BOOL;
   POS_01_Kinetix_01 : BOOL;
   Pos_02_Almacen_2 : BOOL;
   POS_02_Kinetix : BOOL;
   POS_02_Kinetix_01 : BOOL;
   Pos_03_Almacen_2 : BOOL;
   POS_03_Kinetix : BOOL;
   POS_03_Kinetix_01 : BOOL;
   Pos_04_Almacen_2 : BOOL;
   POS_04_Kinetix : BOOL;
   POS_04_Kinetix_01 : BOOL;
   Pos_05_Almacen_2 : BOOL;
   POS_05_Kinetix : BOOL;
   POS_05_Kinetix_01 : BOOL;
   POS_06_Kinetix : BOOL;
   POS_07_Kinetix_Giro : BOOL;
   POS_8 : TIMER := (PRE := 1000, ACC := 887, TT := 1, DN := 1);
   Posicion_4 : BOOL;
   posicion_5 : BOOL := 1;
   PosicionAlmacen : DINT := 128;
   Prensa_Abierta_CNC_1 : BOOL := 1;   // Sensor para Detectar Prensa Abierta CNC 1 Conveyor 1
   Prensa_Presencia_Pieza_CNC_1 : BOOL := 1;   // Sensor para detectar Pieza dentro de la Prensa del CNC 1 Conveyor 1
   Puerta_Abierta_CNC_1 : BOOL := 1;   // Sensor de Puerta Abierta en CNC 1 Conveyor 1
   Pulso : DINT;
   PV_Auto : BOOL := 1;
   PV_Hold : BOOL;
   PV_HomeWh2 : BOOL;
   PV_PosY : DINT := 700;
   PV_SelectedPlace : BOOL := 1;
   PV_SelPlace : DINT := 1;
   PV_Start : BOOL;
   PV_UndoSelect : BOOL;
   PV_Y_Man : BOOL;
   PZA_INICIO : BOOL;
   Rec_Pza_P0_A2 : BOOL;
   Red_Light_Alm_2 : BOOL;
   REG_CHANGER_1 : BOOL;
   REG_CHANGER_2 : BOOL;
   Resert_PF525_From_SFTY : DINT;
   Reset_Almacen_2_PF525_Conv_2 : BOOL;
   Reset_Pasos : BOOL;
   Reset_Pasos_Kinetix : TIMER := (PRE := 2000);
   Reset_ValvulaGeneral_Conv_2 : BOOL;
   RUN_CONV_02 : BOOL;
   run_salida_almacen : BOOL;
   Running_Kinetix : BOOL := 1;
   Running_Kinetix_01 : BOOL;
   Safety_FromTEC81 : Safety := (Connection_Status.RunMode := 1, DINT := 15);
   Safety_OK : BOOL := 1;
   SEMI_END : TIMER := (PRE := 1000);
   SEN_02 : BOOL;
   SEN_IZQ_HOR_OK : BOOL;
   SENS_IZQ_ok : BOOL;
   Sensor_Difuso_1_1_Conv_2 : BOOL;   // Sensor Difuso Presencia Lado A Almacen 1-1
   Sensor_Difuso_1_2_Conv_2 : BOOL;   // Sensor Difuso Presencia Lado A Almacén 1-2
   Sensor_Difuso_2_1_Conv_2 : BOOL;   // Sensor Difuso Presencia Lado B CNC 2-1
   Sensor_Difuso_2_2_Conv_2 : BOOL;   // Sensor Difuso Presencia Lado B CNC 2-2
   Sensor_Difuso_3_1_Conv_2 : BOOL;   // Sensor Difuso Presencia Lado A CNC 3-1
   Sensor_Difuso_3_2_Conv_2 : BOOL;   // Sensor Difuso Presencia Lado A CNC 3-2
   Sensor_Inductivo_Alimentacion_Conv_1 : BOOL;   // Sensor Inductivo Alimentacion y Salida Almacen Conveyor 1
   Sensor_Inductivo_Alimentacion_Conv_2 : BOOL;   // Sensor Inductivo a Salida/entrada Almacen
   Sensor_Inductivo_Almacen_Conv_2 : BOOL;   // Sensor Inductivo Lado A Almacén (Entrada)
   Sensor_Inductivo_CNC_2_Conv_2 : BOOL;   // Sensor Inductivo Posición Lado A CNC
   Sensor_Inductivo_CNC_Conv_2 : BOOL;   // Sensor Inductivo Posición Lado B CNC
   Sensor_Inductivo_Entrada_Conv_1 : BOOL;   // Sensor Inductivo Entrada Lado CNC (Adelante)
   Sensor_Inductivo_Entrada_Conv_2 : BOOL;   // Sensor Inductivo Lado B CNC (Entrada) Conveyor 2
   Sensor_Inductivo_Limit_Conv_2 : BOOL;   // Sensor Inductivo Limit Switch (Revisarl, Empate)
   Sensor_Inductivo_Vision_Conv_2 : BOOL;   // Sensor Presencia Zona de Marcadora Láser
   Sensor_Limit_Up_Conv_2 : BOOL;   // Limit Switch Arriba
   Sensor_PH_Ext_Conv_1 : BOOL;   // Sensor Pistón Horizontal Extendido
   Sensor_PH_Ext_Conv_2 : BOOL;   // Sensor Pistón Horizontal Extendido
   Sensor_PH_Ret_Conv_1 : BOOL := 1;   // Sensor Pistón Horizontal Retraido
   Sensor_PH_Ret_Conv_2 : BOOL := 1;   // Sensor Pistón Horizontal Retraido
   Sensor_Tope_CNC_Conv_2 : BOOL;   // Sensor Tope Pistón CNC
   Sensor_Tope_Marcadora_Conv_1 : BOOL;   // Sensor Pistón Tope Marcadora Láser
   Sensor_Tope_Marcadora_Conv_2 : BOOL;   // Sensor Pistón Tope Marcadora Láser
   Sensor_Tope_PH_Conv_1 : BOOL;   // Sensor Tope Pistón Horizontal
   Sensor_Tope_PH_Conv_2 : BOOL;   // Sensor Tope Pistón Horizontal (Salida de Conveyor 2)
   Sensor_Tope_Vision_Conv_2 : BOOL;   // Sensor Pistón Tope Cámara de Visión
   Sequence_Mover_A_Marcadora_Conv_2 : BOOL;
   Sequence_MoverACamara_Conv_2 : BOOL;
   Sequence_Start_Conv_2 : BOOL;
   Sfty_OK : BOOL := 1;
   Signal_Fanuc_Tomar_Pieza_Conv_2 : BOOL;
   Signal_Marcadora_Conv_2 : BOOL;
   Slector_Automatico_Conv_2 : BOOL := 1;
   Start_Almacen_1_PF525_Conv_2 : BOOL;
   START_CON_STOP_1 : BOOL;
   START_CON_STOP_2 : TIMER := (PRE := 500);
   Start_Conv_1_ONS : BOOL := 1;
   Start_Conv_2 : BOOL;
   Start_Kinetix_Alm_2 : DINT; {produced}
   Start_Motor_Alm_2 : BOOL;
   Start_Rec_PO_A2 : BOOL;
   Start_Warehouse_2 : BOOL;
   stat_test_motor : BOOL := 1;
   STAY_ON_STOP_2 : BOOL;
   STAY_ON_T_STAY : BOOL;
   Step0 : BOOL := 1;   // Condiciones iniciales
   Step1 : BOOL;   // Y to Y Pick
   Step10 : BOOL;   // Open Gripper
   Step11 : BOOL;   // Y to Y place safe
   step12 : BOOL;   // Z to Z2
   step13 : BOOL;   // Esperar Pieza Terminada
   Step14 : BOOL;   // Y to Y place
   Step15 : BOOL;   // Z to Z1
   Step16 : BOOL;   // Close Gripper
   Step17 : BOOL;   // Y to Y PlaceOffset
   Step18 : BOOL;   // S t o S1
   Step19 : BOOL;   // X to X2
   Step2 : BOOL;   // X to X1
   Step20 : BOOL;   // Y to Y PickOffset
   Step21 : BOOL;   // Z to Z2
   Step22 : BOOL;   // Y to Y Pick
   Step23 : BOOL;   // Open Gripper
   Step24 : BOOL;   // Y to Y Pcik Safe
   Step25 : BOOL;   // Z to Z1
   Step26 : BOOL;   // Homming
   Step27 : BOOL;
   Step28 : BOOL;
   Step29 : BOOL;
   Step3 : BOOL;   // Z to Z2
   Step30 : BOOL;
   Step4 : BOOL;   // Close Gripper
   Step5 : BOOL;   // Y to Y PickOffset
   Step6 : BOOL;   // Z to Z1
   Step7 : BOOL;   // Y to Y PlaceOffset
   Step8 : BOOL;   // S to S2
   step9 : BOOL;   // Y to Y Place
   Step_00_Conv_1 : BOOL;
   Step_00_Conv_2 : BOOL := 1;
   Step_01_Conv_1 : BOOL;
   Step_01_Conv_2 : BOOL;
   Step_02_Conv_1 : BOOL;
   Step_02_Conv_2 : BOOL;
   Step_03_Conv_1 : BOOL;
   Step_03_Conv_2 : BOOL;
   Step_04_Conv_1 : BOOL;
   Step_04_Conv_2 : BOOL;
   Step_05_Conv_1 : BOOL;
   Step_05_Conv_2 : BOOL;
   Step_06_Conv_1 : BOOL;
   Step_06_Conv_2 : BOOL;   // Step 25 *** Cambio de Dirección de Pieza para regresar, activa Pistón, espera señalde pistón lateral Extendido ***
   Step_07_Conv_1 : BOOL;
   Step_07_Conv_2 : BOOL;
   Step_08_Conv_1 : BOOL;
   Step_08_Conv_2 : BOOL;
   Step_09_Conv_1 : BOOL;
   Step_09_Conv_2 : BOOL;
   Step_10_Conv_1 : BOOL;
   Step_10_Conv_2 : BOOL;
   Step_11_Conv_1 : BOOL;
   Step_11_Conv_2 : BOOL;
   Step_12_Conv_1 : BOOL;
   Step_12_Conv_2 : BOOL;
   Step_13_Conv_1 : BOOL;
   Step_13_Conv_2 : BOOL;
   Step_14_Conv_1 : BOOL;
   Step_14_Conv_2 : BOOL;
   Step_15_Conv_1 : BOOL;
   Step_15_Conv_2 : BOOL;
   Step_16_Conv_1 : BOOL;
   Step_16_Conv_2 : BOOL;
   Step_17_Conv_1 : BOOL;
   Step_17_Conv_2 : BOOL;
   Step_18_Conv_1 : BOOL;
   Step_18_Conv_2 : BOOL;
   Step_19_Conv_1 : BOOL;
   Step_19_Conv_2 : BOOL;
   Step_20_Conv_1 : BOOL;
   Step_20_Conv_2 : BOOL;
   Step_21_Conv_1 : BOOL;
   Step_21_Conv_2 : BOOL;
   Step_22_Conv_1 : BOOL;
   Step_23_Conv_1 : BOOL;
   Step_24_Conv_1 : BOOL := 1;
   Step_25_Conv_1 : BOOL;
   Step_26_Conv_1 : BOOL;
   Step_27_Conv_1 : BOOL;
   Step_28_Conv_1 : BOOL;
   Step_29_Conv_1 : BOOL;
   Step_30_Conv_1 : BOOL;
   Step_31_Conv_1 : BOOL;
   Step_32_Conv_1 : BOOL;
   Step_33_Conv_1 : BOOL;
   Step_34_Conv_1 : BOOL;
   Step_35_Conv_1 : BOOL;
   Step_36_Conv_1 : BOOL;
   Step_37_Conv_1 : BOOL;
   Step_38_Conv_1 : BOOL;
   Step_39_Conv_1 : BOOL;
   Step_40_Conv_1 : BOOL;
   STOP_2 : TIMER := (PRE := 500);
   Stop_Kinetix : BOOL;
   STOP_STOPER_2 : BOOL;
   StorageSeqToTec81 : DINT := 130; {produced}
   T_Conv_1_Sin_Pieza : TIMER := (PRE := 60000);
   T_Conv_2_Stop_Last_Time : TIMER := (PRE := 2500);
   T_Intermedio_Alm_2 : TIMER := (PRE := 500, ACC := 500, EN := 1, DN := 1);
   T_Permisive_Step_00 : TIMER := (PRE := 150);
   T_Permisive_Step_01 : TIMER := (PRE := 150);
   T_Permisive_Step_02 : TIMER := (PRE := 150);
   T_Permisive_Step_03 : TIMER := (PRE := 150);
   T_Permisive_Step_04 : TIMER := (PRE := 500);
   T_Permisive_Step_05 : TIMER := (PRE := 150);
   T_Permisive_Step_06 : TIMER := (PRE := 150);
   T_Permisive_Step_07 : TIMER := (PRE := 150);
   T_Permisive_Step_08 : TIMER := (PRE := 150);
   T_Permisive_Step_09 : TIMER := (PRE := 150);
   T_Permisive_Step_10 : TIMER := (PRE := 150);
   T_Permisive_Step_11 : TIMER := (PRE := 150);
   T_Permisive_Step_12 : TIMER := (PRE := 150);
   T_Permisive_Step_13 : TIMER := (PRE := 150);
   T_Permisive_Step_14 : TIMER := (PRE := 150);
   T_Permisive_Step_15 : TIMER := (PRE := 150);
   T_Permisive_Step_16 : TIMER := (PRE := 150);
   T_Permisive_Step_17 : TIMER := (PRE := 150);
   T_Permisive_Step_18 : TIMER := (PRE := 150);
   T_Permisive_Step_19 : TIMER := (PRE := 150);
   T_Permisive_Step_20 : TIMER := (PRE := 150);
   T_Permisive_Step_21 : TIMER := (PRE := 150);
   T_Permisive_Step_22 : TIMER := (PRE := 150);
   T_Permisive_Step_23 : TIMER := (PRE := 150);
   T_Permisive_Step_24 : TIMER := (PRE := 150);
   T_Permisive_Step_25 : TIMER := (PRE := 150);
   T_Permisive_Step_26 : TIMER := (PRE := 150);
   T_Permisive_Step_27 : TIMER := (PRE := 150);
   T_Permisive_Step_28 : TIMER := (PRE := 150);
   T_Permisive_Step_29 : TIMER := (PRE := 150);
   T_Permisive_Step_30 : TIMER := (PRE := 150);
   T_Permisive_Step_31 : TIMER := (PRE := 150);
   T_Permisive_Step_32 : TIMER := (PRE := 150);
   T_Permisive_Step_33 : TIMER := (PRE := 150);
   T_Permisive_Step_34 : TIMER := (PRE := 150);
   T_Permisive_Step_35 : TIMER := (PRE := 150);
   T_Permisive_Step_36 : TIMER := (PRE := 150);
   T_Permisive_Step_37 : TIMER := (PRE := 150);
   T_Permisive_Step_38 : TIMER := (PRE := 150);
   T_Permisive_Step_39 : TIMER := (PRE := 150);
   T_Permisive_Step_40 : TIMER := (PRE := 150);
   T_Permissive_HomeStep0 : BOOL;
   T_Permissive_HomeStep1 : TIMER := (PRE := 2000);
   T_Permissive_HomeStep2 : TIMER := (PRE := 150);
   T_Permissive_HomeStep3 : TIMER := (PRE := 150);
   T_Permissive_HomeStep4 : TIMER := (PRE := 150);
   T_Permissive_HomeStep5 : TIMER := (PRE := 150);
   T_Permissive_HomeStep6 : TIMER := (PRE := 150);
   T_Permissive_HomeStep7 : TIMER := (PRE := 150);
   T_Permissive_HomeStep8 : TIMER := (PRE := 150);
   T_Permissive_HomeStep9 : TIMER := (PRE := 500);
   T_Permissive_HomStep0 : TIMER := (PRE := 1500);
   T_Permissive_Step0 : TIMER := (PRE := 150);
   T_Permissive_Step1 : TIMER := (PRE := 150);
   T_Permissive_Step10 : TIMER := (PRE := 150);
   T_Permissive_Step11 : TIMER := (PRE := 150);
   T_Permissive_Step12 : TIMER := (PRE := 150);
   T_Permissive_Step13 : TIMER := (PRE := 150);
   T_Permissive_Step14 : TIMER := (PRE := 150);
   T_Permissive_Step15 : TIMER := (PRE := 150);
   T_Permissive_Step16 : TIMER := (PRE := 150);
   T_Permissive_Step17 : TIMER := (PRE := 150);
   T_Permissive_Step18 : TIMER := (PRE := 150);
   T_Permissive_Step19 : TIMER := (PRE := 150);
   T_Permissive_Step2 : TIMER := (PRE := 150);
   T_Permissive_Step20 : TIMER := (PRE := 150);
   T_Permissive_Step21 : TIMER := (PRE := 150);
   T_Permissive_Step22 : TIMER := (PRE := 150);
   T_Permissive_Step23 : TIMER := (PRE := 150);
   T_Permissive_Step24 : TIMER := (PRE := 150);
   T_Permissive_Step25 : TIMER := (PRE := 150);
   T_Permissive_Step26 : TIMER;
   T_Permissive_Step27 : TIMER;
   T_Permissive_Step28 : TIMER;
   T_Permissive_Step29 : TIMER;
   T_Permissive_Step3 : TIMER := (PRE := 150);
   T_Permissive_Step30 : TIMER;
   T_Permissive_Step4 : TIMER := (PRE := 500);
   T_Permissive_Step5 : TIMER := (PRE := 150);
   T_Permissive_Step6 : TIMER := (PRE := 150);
   T_Permissive_Step7 : TIMER := (PRE := 150);
   T_Permissive_Step8 : TIMER := (PRE := 150);
   T_Permissive_Step9 : TIMER := (PRE := 150);
   T_Pieza_Antes_Marcadora : TIMER := (PRE := 1000);
   T_Pieza_FinDeCarrera_Conv_2 : TIMER := (PRE := 3000);
   T_Pieza_FinDeCarrera_Error_Conv_2 : TIMER := (PRE := 3000);
   T_Pieza_FinDeCarrera_Salida : TIMER := (PRE := 10000);
   T_Pieza_Marcadora : TIMER := (PRE := 20000);
   T_Pieza_Marcadora_Conv_2 : TIMER := (PRE := 3000);
   T_Pieza_MarcadoraTerminada_Conv_2 : TIMER := (PRE := 10000);
   T_Pieza_TomaFanuc_Conv_2 : TIMER := (PRE := 3000);
   Tec81_to_Wh2 : DINT;
   Test : INT := 1;
   Test_Bit : DINT := -1879048191;
   Test_leaa : DINT := 1;
   Time_out_Conv_2 : TIMER := (PRE := 30000);
   TIMER0 : TIMER := (PRE := 5000);
   TIMER_1 : TIMER := (PRE := 3000);
   TIMER_22 : TIMER := (PRE := 3000);
   TIMER_FINAL : TIMER := (PRE := 6000, ACC := 6000);
   TIMER_OFF_STOP : TIMER := (PRE := 500);
   timer_piston_2 : TIMER := (PRE := 1500);
   timer_piston_3 : TIMER := (PRE := 1500);
   TIMER_READY_STOP : TIMER := (PRE := 5000);
   timer_salida_plato : TIMER := (PRE := 3000, ACC := 3000, EN := 1, DN := 1);
   TIMER_START_CON : TIMER := (PRE := 500);
   TIMER_STOP_1 : TIMER := (PRE := 5000);
   TIMER_STOP_2 : TIMER := (PRE := 13000);
   TIMER_X : TIMER := (PRE := 500);
   TMR10_CONV_02 : TIMER := (PRE := 1500);
   TMR20 : TIMER := (PRE := 1000);
   TMR21 : TIMER := (PRE := 2000);
   TMR_01 : TIMER := (PRE := 1000);
   TMR_02 : TIMER := (PRE := 1500);
   tmr_03 : TIMER := (PRE := 2000);
   TMR_04 : TIMER := (PRE := 1500);
   TMR_05 : TIMER := (PRE := 1500);
   TMR_06 : TIMER := (PRE := 1500);
   TMR_07 : TIMER := (PRE := 1500);
   TMR_1 : TIMER := (PRE := 1500);
   TMR_20 : TIMER := (PRE := 1500);
   TMR_CONV01 : TIMER := (PRE := 4000);
   TMR_Esp_Abrir_Griper : TIMER := (PRE := 1500);
   TMR_Esp_Pos_6 : TIMER := (PRE := 1500);
   TMR_Esp_Pos_7 : TIMER := (PRE := 1500);
   TMR_ESPERA : BOOL;
   TMR_Gripper : TIMER := (PRE := 1500);
   TMR_GRIPPER_SALIDA : TIMER := (PRE := 1500);
   Tmr_Pistion_Adelante : TIMER := (PRE := 1500, EN := 1, DN := 1);
   TMR_pos6 : TIMER;
   TMR_POS8 : TIMER := (PRE := 1000);
   Tmr_Pos_6 : TIMER := (PRE := 1000, ACC := 1000, EN := 1, DN := 1);
   TN : DINT;
   TN_FIN_LF : BOOL;
   TN_FIN_LI : BOOL;
   TN_S1 : BOOL;
   TN_STOP_1 : BOOL;
   To_Pos_Alm_2 : DINT := 128; {produced}
   Tomar_pieza : BOOL;
   Tope_CNC_Conv_2 : BOOL;   // Tope Pistón CNC (Freno 5) Conveyor 2
   Tope_Marcadora_Conv_2 : BOOL;   // Tope Pistón Marcadora Láser (Freno 6) Conveyor 2
   Tope_Salida_PH_Conv_2 : BOOL := 1;   // Tope Pistón Salida de Producto (Freno 8) Conveyor 2
   Tope_Vision_Conv_2 : BOOL;   // Tope Pistón Cámara de Visión Conveyor 2
   WAIT : TIMER := (PRE := 3000);
   WAIT_STOP_2 : TIMER := (PRE := 5000);
   Warehouse_2_Actual_Step : DINT := 130;
   Warehouse_2_Step : DINT := 8192;
        .20   // MUEVE SERVO HACIA POSICIÓN PREVIA A DEJAR PIEZA EN ALMACÉN
        .5   // MUEVE SERVO HACIA ARRIBA PARA PODER RETIRAR LA PIEZA LIBREMENTE
        .24   // MUEVE SERVO
        .22   // MUEVE SERVO PARA DEJAR PIEZA EN POSICIÓN FINAL EN ALMACÉN DE SALIDA
        .25   // MUEVE ACTUADOR EJE Z HACIA TRANSPORTADOR
        .26   // ESPERA FINALIZAR SECUENCIA DE HOME
        .7   // MUEVE SERVO HACIA LA POSICIÓN PARA PREVIA A DEJAR PIEZA EN TRASNPORTADOR
        .9   // MUEVE SERVO A ALTURA DE TRANSPORTADOR
        .0   // VERIFICA POSICIÓN INICIAL SEGURA
        .1   // MUEVE SERVO HACIA POSICIÓN SELECCIONADA
        .10   // ABRE GRIPPER
        .11   // MUEVE SERVO DE MANERA SEGURA
        .12   // RETRAE ACTUADOR EJE Z HACIA LADO ALMACÉN
        .13   // ESPERA PIEZA TERMINADA PARA RETORNO A ALMACÉN
        .14   // MUEVE SERVO PARA RECIBIR PIEZA DE TRANSPORTADOR
        .15   // MUEVE ACTUADOR DE EJE Z HACIA TRANSPORTADOR
        .16   // CIERRA GRIPPER
        .17   // SUBE SERVO
        .18   // GIRA ACTUADOR HACIA ALMACÉN
        .19   // MUEVE ACTUADOR EN EJE X HACIA SALIDA DE ALMACÉN
        .3   // MUEVE ACTUADOR EJE Z HACIA TOMA DE PIEZA EN ALMACÉN
        .4   // CIERRA GRIPPER
        .2   // MUEVE ACTUADOR EJE X HACIA LADO DE TOMA DE PIEZA EN ALMACÉN
        .6   // RETRAE ACTUADOR PARA SACAR PIEZA DE ALMACÉN
        .21   // MUEVE ACTUADOR EJE Z HACIA ALMACÉN
        .8   // GIRA ACTUADOR HACIA TRANSPORTADOR
        .23   // ABRE GRIPPER
   Wh2_GripperClosed : BOOL;
   Wh2_GripperOpen : BOOL;
   Wh2_Matrix : DINT[32] := ([1] := 895, [2] := 715, [3] := 535, [4] := 355, [5] := 175, [14] := 380, [15] := 338);
   Wh2_to_Tec81 : DINT := 4; {produced}
   Wh2_X1 : BOOL;   // Posición de toma de pieza en eje X
   Wh2_Y : DINT[16];
   Wh2_YActualPosition : REAL := 439.95758;
   Wh2_Z1 : BOOL := 1;
   Wh2_Z2 : BOOL;
   Wh_2_Home_Actual_Step : DINT;
   Wh_2_Home_Step : BOOL;
   Wh_2_HomeSeq_Perm_OnDly : TIMER[16] := ([2].PRE := 100, [3].PRE := 100, [4].PRE := 100, [5].PRE := 100, [6].PRE := 100, [7].PRE := 100, [8].PRE := 100, [9].PRE := 100);
   Wh_2_Homming_Step : DINT := 1;
        .3   // GIRA ACTUADOR
        .4   // MUEVE SERVO A HOME
        .0   // SOLICITUD DE HOME
        .9   // HOME TERMINADO
        .5   // MUEVE ACTUDOR EJE Z
        .1   // EVALUA LAS CONDICIONES ACTUALES ANTES DE PROSEGUIR
        .6   // GIRA GRIPPER
        .7   // MUEVE ACTUADOR EJE X
        .8   // ABRE GRIPPER
        .2   // GIRA ACTUADOR
   Wh_2_Perm_OnDly : TIMER[32] := ([0].PRE := 100, [1].PRE := 100, [2].PRE := 100, [3].PRE := 100, [4].PRE := 100, [5].PRE := 100, [6].PRE := 100, [7].PRE := 100, [8].PRE := 100, [9].PRE := 100, [10].PRE := 100, [11].PRE := 100, [12].PRE := 100, [13].PRE := 100, [14].PRE := 100, [15].PRE := 100, [16].PRE := 100, [17].PRE := 100, [18].PRE := 100, [19].PRE := 100, [20].PRE := 100, [21].PRE := 100, [22].PRE := 100, [23].PRE := 100, [24].PRE := 100, [25].PRE := 100, [26].PRE := 100);
   Wh_2_X : DINT; {produced}
   Wh_2_Y : DINT := 380; {produced}   // Posición de almacén en eje Y
   Wh_S1 : BOOL := 1;
   Yellow_Light_Alm_2 : BOOL;
   YSafePos : BOOL;
END_VAR

PROGRAM MainProgram   (* main routine Prueba *)
VAR
   ACT1 : BOOL;
   Contador_Stop_Conveyor : COUNTER := (PRE := 4);
   OS1 : BOOL;
   PosDer_Alm_0_C : BOOL;
   PosDer_Alm_0_E : BOOL;
   PosDer_Alm_1_C : BOOL;
   PosDer_Alm_1_E : BOOL;
   PosDer_Alm_2_C : BOOL;
   PosDer_Alm_2_E : BOOL;
   PosDer_Alm_3_C : BOOL;
   PosDer_Alm_3_E : BOOL;
   PosDer_Alm_4_C : BOOL;
   PosDer_Alm_4_E : BOOL;
   PosDer_Alm_5_C : BOOL;
   PosDer_Alm_5_E : BOOL;
   PosIzq_Alm_0_C : BOOL;
   PosIzq_Alm_0_E : BOOL;
   PosIzq_Alm_1_C : BOOL;
   PosIzq_Alm_1_E : BOOL;
   PosIzq_Alm_2_C : BOOL;
   PosIzq_Alm_2_E : BOOL;
   PosIzq_Alm_3_C : BOOL;
   PosIzq_Alm_3_E : BOOL;
   PosIzq_Alm_4_C : BOOL;
   PosIzq_Alm_4_E : BOOL;
   PosIzq_Alm_5_C : BOOL;
   PosIzq_Alm_5_E : BOOL;
   PosIzq_Alm_7_C : BOOL;
   PosIzq_Conv_7_C : BOOL;
   PosIzq_Conv_8_C : BOOL;
   PosProgramming : BOOL;
   SEN1 : BOOL;
   Start_Conveyor_2 : BOOL;
   Start_Rutine : BOOL;
   Stop_Conveyor_2 : BOOL;
   tag_switch : BOOL;
   tag_switch2 : BOOL;
   tag_switch3 : BOOL;
   Tag_switch4 : BOOL;
   tag_timer_piston : BOOL;
   tag_timer_piston2 : BOOL;
   tag_timer_piston3 : BOOL;
   Timer1 : TIMER := (PRE := 3000);
   Timer2 : TIMER := (PRE := 3000);
   Timer3 : TIMER := (PRE := 6000);
   Timer4 : TIMER := (PRE := 13000);
   Timer5 : TIMER := (PRE := 4000);
   Timer6 : TIMER := (PRE := 5000);
   Timer7 : TIMER := (PRE := 3000);
END_VAR

ROUTINE Almacen2   (* ladder *)
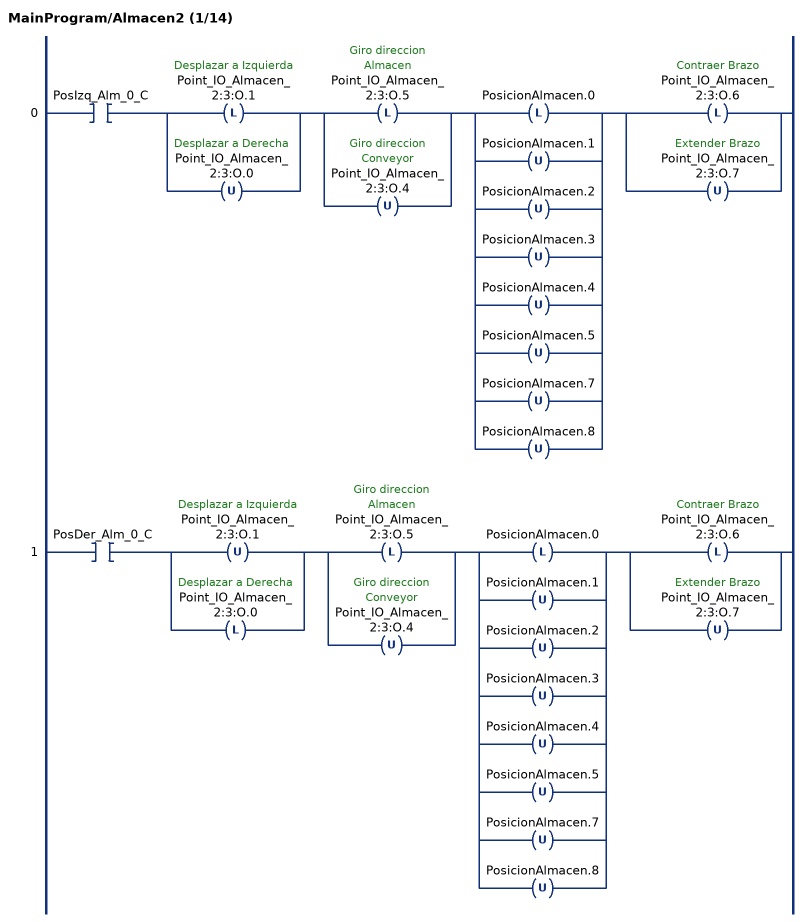
   0: XIC(PosIzq_Alm_0_C)[OTL(Point_IO_Almacen_2:3:O.1) ,OTU(Point_IO_Almacen_2:3:O.0) ][OTL(Point_IO_Almacen_2:3:O.5) ,OTU(Point_IO_Almacen_2:3:O.4) ][OTL(PosicionAlmacen.0) ,OTU(PosicionAlmacen.1) ,OTU(PosicionAlmacen.2) ,OTU(PosicionAlmacen.3) ,OTU(PosicionAlmacen.4) ,OTU(PosicionAlmacen.5) ,OTU(PosicionAlmacen.7) ,OTU(PosicionAlmacen.8) ][OTL(Point_IO_Almacen_2:3:O.6) ,OTU(Point_IO_Almacen_2:3:O.7) ];
   1: XIC(PosDer_Alm_0_C)[OTU(Point_IO_Almacen_2:3:O.1) ,OTL(Point_IO_Almacen_2:3:O.0) ][OTL(Point_IO_Almacen_2:3:O.5) ,OTU(Point_IO_Almacen_2:3:O.4) ][OTL(PosicionAlmacen.0) ,OTU(PosicionAlmacen.1) ,OTU(PosicionAlmacen.2) ,OTU(PosicionAlmacen.3) ,OTU(PosicionAlmacen.4) ,OTU(PosicionAlmacen.5) ,OTU(PosicionAlmacen.7) ,OTU(PosicionAlmacen.8) ][OTL(Point_IO_Almacen_2:3:O.6) ,OTU(Point_IO_Almacen_2:3:O.7) ];
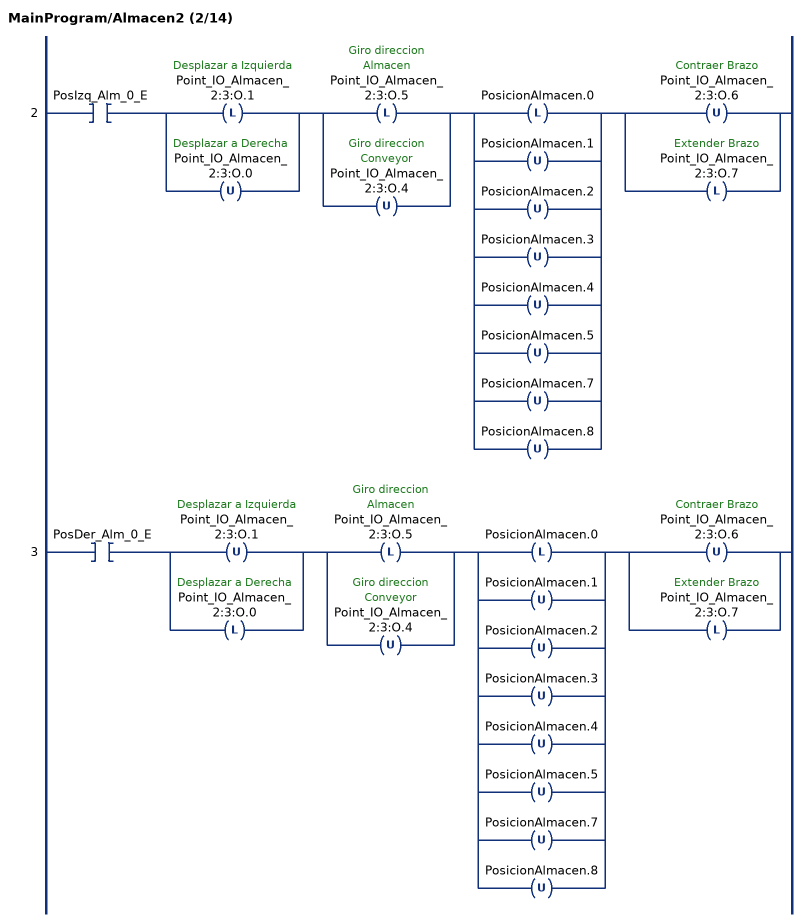
   2: XIC(PosIzq_Alm_0_E)[OTL(Point_IO_Almacen_2:3:O.1) ,OTU(Point_IO_Almacen_2:3:O.0) ][OTL(Point_IO_Almacen_2:3:O.5) ,OTU(Point_IO_Almacen_2:3:O.4) ][OTL(PosicionAlmacen.0) ,OTU(PosicionAlmacen.1) ,OTU(PosicionAlmacen.2) ,OTU(PosicionAlmacen.3) ,OTU(PosicionAlmacen.4) ,OTU(PosicionAlmacen.5) ,OTU(PosicionAlmacen.7) ,OTU(PosicionAlmacen.8) ][OTU(Point_IO_Almacen_2:3:O.6) ,OTL(Point_IO_Almacen_2:3:O.7) ];
   3: XIC(PosDer_Alm_0_E)[OTU(Point_IO_Almacen_2:3:O.1) ,OTL(Point_IO_Almacen_2:3:O.0) ][OTL(Point_IO_Almacen_2:3:O.5) ,OTU(Point_IO_Almacen_2:3:O.4) ][OTL(PosicionAlmacen.0) ,OTU(PosicionAlmacen.1) ,OTU(PosicionAlmacen.2) ,OTU(PosicionAlmacen.3) ,OTU(PosicionAlmacen.4) ,OTU(PosicionAlmacen.5) ,OTU(PosicionAlmacen.7) ,OTU(PosicionAlmacen.8) ][OTU(Point_IO_Almacen_2:3:O.6) ,OTL(Point_IO_Almacen_2:3:O.7) ];
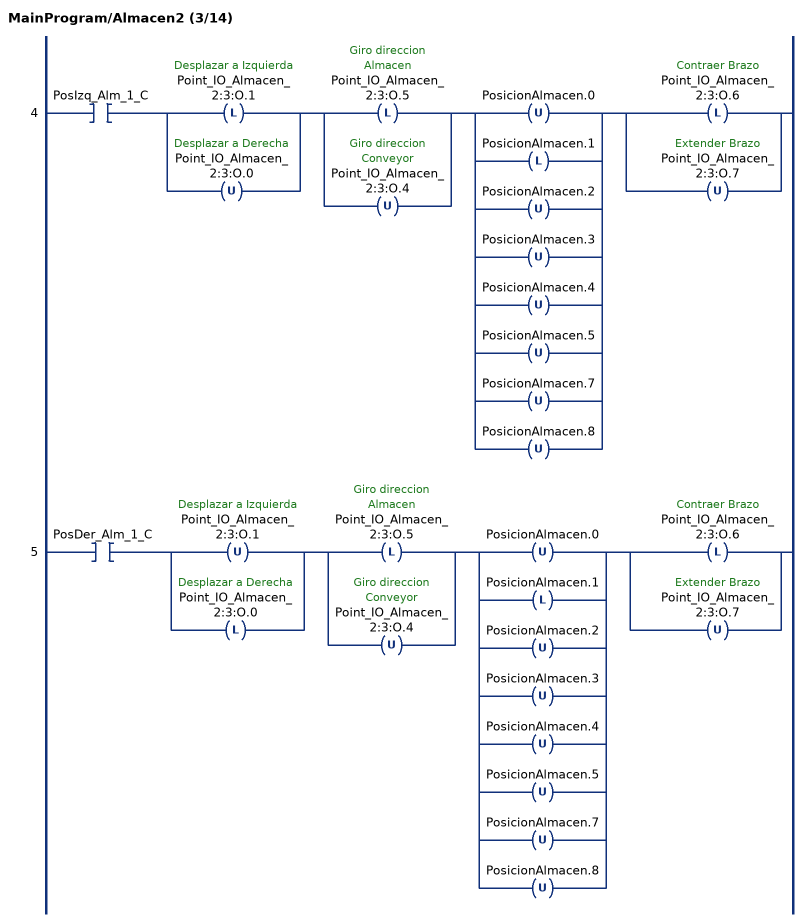
   4: XIC(PosIzq_Alm_1_C)[OTL(Point_IO_Almacen_2:3:O.1) ,OTU(Point_IO_Almacen_2:3:O.0) ][OTL(Point_IO_Almacen_2:3:O.5) ,OTU(Point_IO_Almacen_2:3:O.4) ][OTU(PosicionAlmacen.0) ,OTL(PosicionAlmacen.1) ,OTU(PosicionAlmacen.2) ,OTU(PosicionAlmacen.3) ,OTU(PosicionAlmacen.4) ,OTU(PosicionAlmacen.5) ,OTU(PosicionAlmacen.7) ,OTU(PosicionAlmacen.8) ][OTL(Point_IO_Almacen_2:3:O.6) ,OTU(Point_IO_Almacen_2:3:O.7) ];
   5: XIC(PosDer_Alm_1_C)[OTU(Point_IO_Almacen_2:3:O.1) ,OTL(Point_IO_Almacen_2:3:O.0) ][OTL(Point_IO_Almacen_2:3:O.5) ,OTU(Point_IO_Almacen_2:3:O.4) ][OTU(PosicionAlmacen.0) ,OTL(PosicionAlmacen.1) ,OTU(PosicionAlmacen.2) ,OTU(PosicionAlmacen.3) ,OTU(PosicionAlmacen.4) ,OTU(PosicionAlmacen.5) ,OTU(PosicionAlmacen.7) ,OTU(PosicionAlmacen.8) ][OTL(Point_IO_Almacen_2:3:O.6) ,OTU(Point_IO_Almacen_2:3:O.7) ];
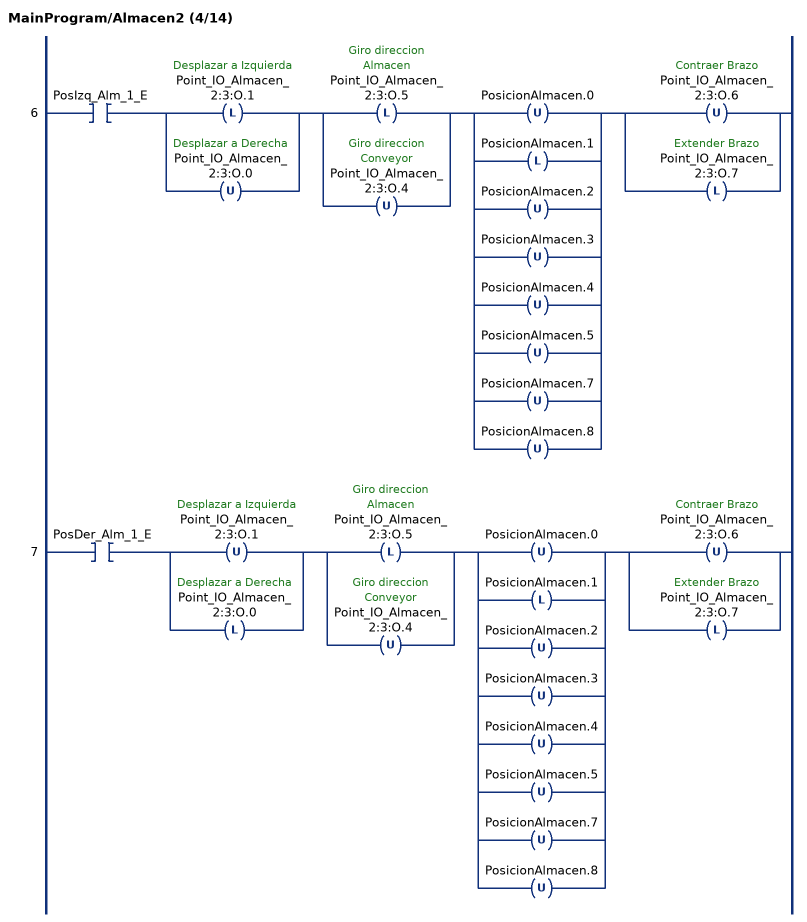
   6: XIC(PosIzq_Alm_1_E)[OTL(Point_IO_Almacen_2:3:O.1) ,OTU(Point_IO_Almacen_2:3:O.0) ][OTL(Point_IO_Almacen_2:3:O.5) ,OTU(Point_IO_Almacen_2:3:O.4) ][OTU(PosicionAlmacen.0) ,OTL(PosicionAlmacen.1) ,OTU(PosicionAlmacen.2) ,OTU(PosicionAlmacen.3) ,OTU(PosicionAlmacen.4) ,OTU(PosicionAlmacen.5) ,OTU(PosicionAlmacen.7) ,OTU(PosicionAlmacen.8) ][OTU(Point_IO_Almacen_2:3:O.6) ,OTL(Point_IO_Almacen_2:3:O.7) ];
   7: XIC(PosDer_Alm_1_E)[OTU(Point_IO_Almacen_2:3:O.1) ,OTL(Point_IO_Almacen_2:3:O.0) ][OTL(Point_IO_Almacen_2:3:O.5) ,OTU(Point_IO_Almacen_2:3:O.4) ][OTU(PosicionAlmacen.0) ,OTL(PosicionAlmacen.1) ,OTU(PosicionAlmacen.2) ,OTU(PosicionAlmacen.3) ,OTU(PosicionAlmacen.4) ,OTU(PosicionAlmacen.5) ,OTU(PosicionAlmacen.7) ,OTU(PosicionAlmacen.8) ][OTU(Point_IO_Almacen_2:3:O.6) ,OTL(Point_IO_Almacen_2:3:O.7) ];
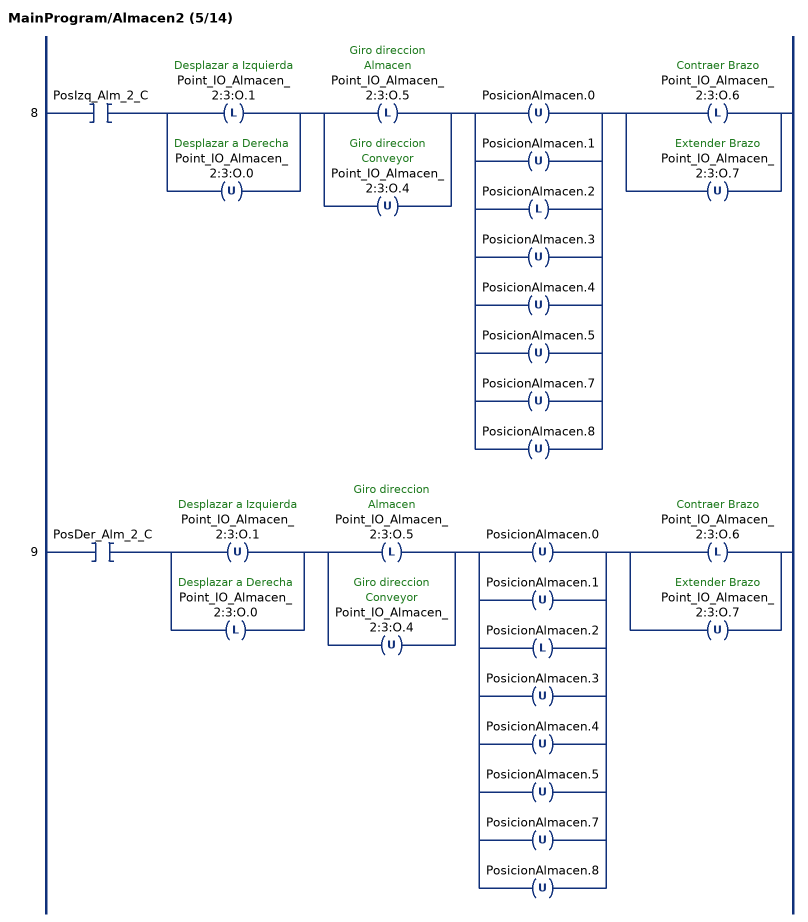
   8: XIC(PosIzq_Alm_2_C)[OTL(Point_IO_Almacen_2:3:O.1) ,OTU(Point_IO_Almacen_2:3:O.0) ][OTL(Point_IO_Almacen_2:3:O.5) ,OTU(Point_IO_Almacen_2:3:O.4) ][OTU(PosicionAlmacen.0) ,OTU(PosicionAlmacen.1) ,OTL(PosicionAlmacen.2) ,OTU(PosicionAlmacen.3) ,OTU(PosicionAlmacen.4) ,OTU(PosicionAlmacen.5) ,OTU(PosicionAlmacen.7) ,OTU(PosicionAlmacen.8) ][OTL(Point_IO_Almacen_2:3:O.6) ,OTU(Point_IO_Almacen_2:3:O.7) ];
   9: XIC(PosDer_Alm_2_C)[OTU(Point_IO_Almacen_2:3:O.1) ,OTL(Point_IO_Almacen_2:3:O.0) ][OTL(Point_IO_Almacen_2:3:O.5) ,OTU(Point_IO_Almacen_2:3:O.4) ][OTU(PosicionAlmacen.0) ,OTU(PosicionAlmacen.1) ,OTL(PosicionAlmacen.2) ,OTU(PosicionAlmacen.3) ,OTU(PosicionAlmacen.4) ,OTU(PosicionAlmacen.5) ,OTU(PosicionAlmacen.7) ,OTU(PosicionAlmacen.8) ][OTL(Point_IO_Almacen_2:3:O.6) ,OTU(Point_IO_Almacen_2:3:O.7) ];
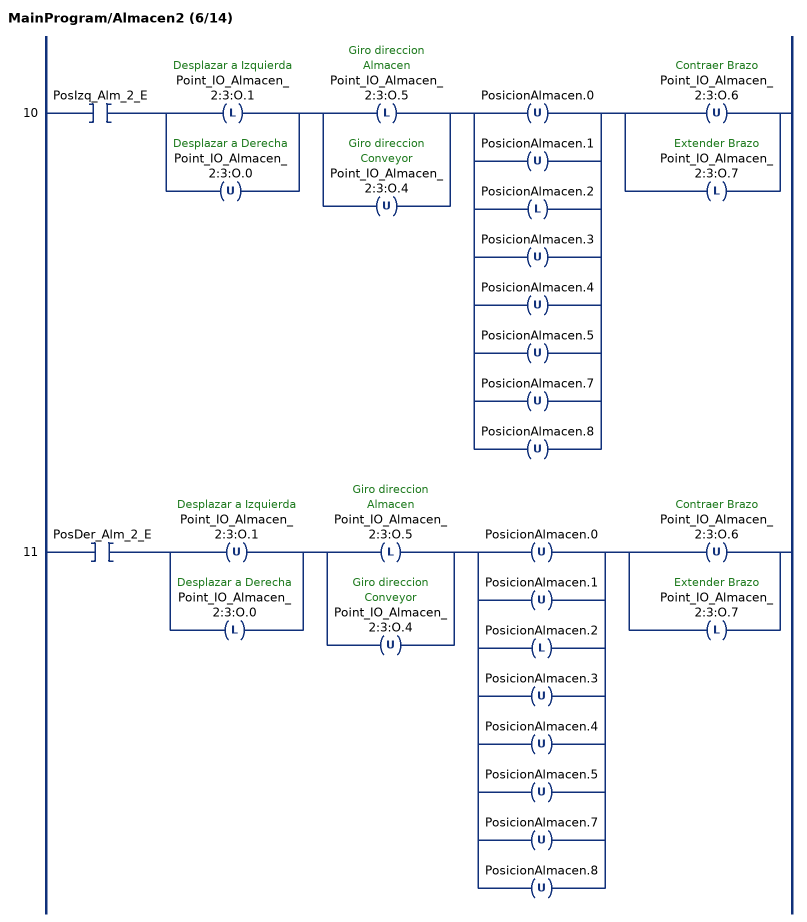
   10: XIC(PosIzq_Alm_2_E)[OTL(Point_IO_Almacen_2:3:O.1) ,OTU(Point_IO_Almacen_2:3:O.0) ][OTL(Point_IO_Almacen_2:3:O.5) ,OTU(Point_IO_Almacen_2:3:O.4) ][OTU(PosicionAlmacen.0) ,OTU(PosicionAlmacen.1) ,OTL(PosicionAlmacen.2) ,OTU(PosicionAlmacen.3) ,OTU(PosicionAlmacen.4) ,OTU(PosicionAlmacen.5) ,OTU(PosicionAlmacen.7) ,OTU(PosicionAlmacen.8) ][OTU(Point_IO_Almacen_2:3:O.6) ,OTL(Point_IO_Almacen_2:3:O.7) ];
   11: XIC(PosDer_Alm_2_E)[OTU(Point_IO_Almacen_2:3:O.1) ,OTL(Point_IO_Almacen_2:3:O.0) ][OTL(Point_IO_Almacen_2:3:O.5) ,OTU(Point_IO_Almacen_2:3:O.4) ][OTU(PosicionAlmacen.0) ,OTU(PosicionAlmacen.1) ,OTL(PosicionAlmacen.2) ,OTU(PosicionAlmacen.3) ,OTU(PosicionAlmacen.4) ,OTU(PosicionAlmacen.5) ,OTU(PosicionAlmacen.7) ,OTU(PosicionAlmacen.8) ][OTU(Point_IO_Almacen_2:3:O.6) ,OTL(Point_IO_Almacen_2:3:O.7) ];
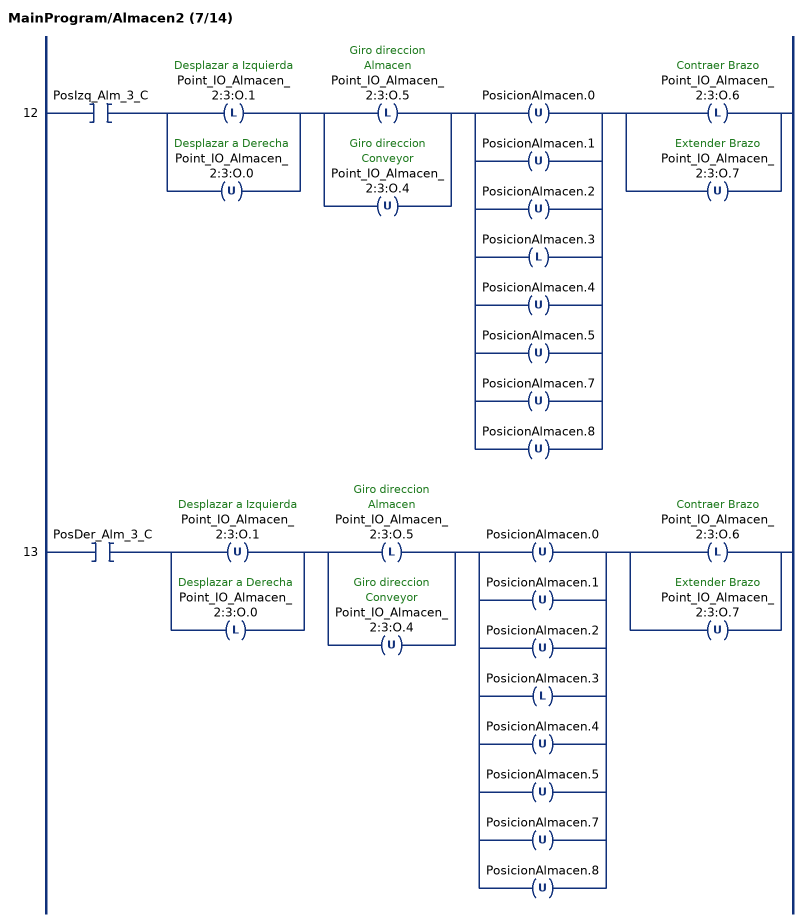
   12: XIC(PosIzq_Alm_3_C)[OTL(Point_IO_Almacen_2:3:O.1) ,OTU(Point_IO_Almacen_2:3:O.0) ][OTL(Point_IO_Almacen_2:3:O.5) ,OTU(Point_IO_Almacen_2:3:O.4) ][OTU(PosicionAlmacen.0) ,OTU(PosicionAlmacen.1) ,OTU(PosicionAlmacen.2) ,OTL(PosicionAlmacen.3) ,OTU(PosicionAlmacen.4) ,OTU(PosicionAlmacen.5) ,OTU(PosicionAlmacen.7) ,OTU(PosicionAlmacen.8) ][OTL(Point_IO_Almacen_2:3:O.6) ,OTU(Point_IO_Almacen_2:3:O.7) ];
   13: XIC(PosDer_Alm_3_C)[OTU(Point_IO_Almacen_2:3:O.1) ,OTL(Point_IO_Almacen_2:3:O.0) ][OTL(Point_IO_Almacen_2:3:O.5) ,OTU(Point_IO_Almacen_2:3:O.4) ][OTU(PosicionAlmacen.0) ,OTU(PosicionAlmacen.1) ,OTU(PosicionAlmacen.2) ,OTL(PosicionAlmacen.3) ,OTU(PosicionAlmacen.4) ,OTU(PosicionAlmacen.5) ,OTU(PosicionAlmacen.7) ,OTU(PosicionAlmacen.8) ][OTL(Point_IO_Almacen_2:3:O.6) ,OTU(Point_IO_Almacen_2:3:O.7) ];
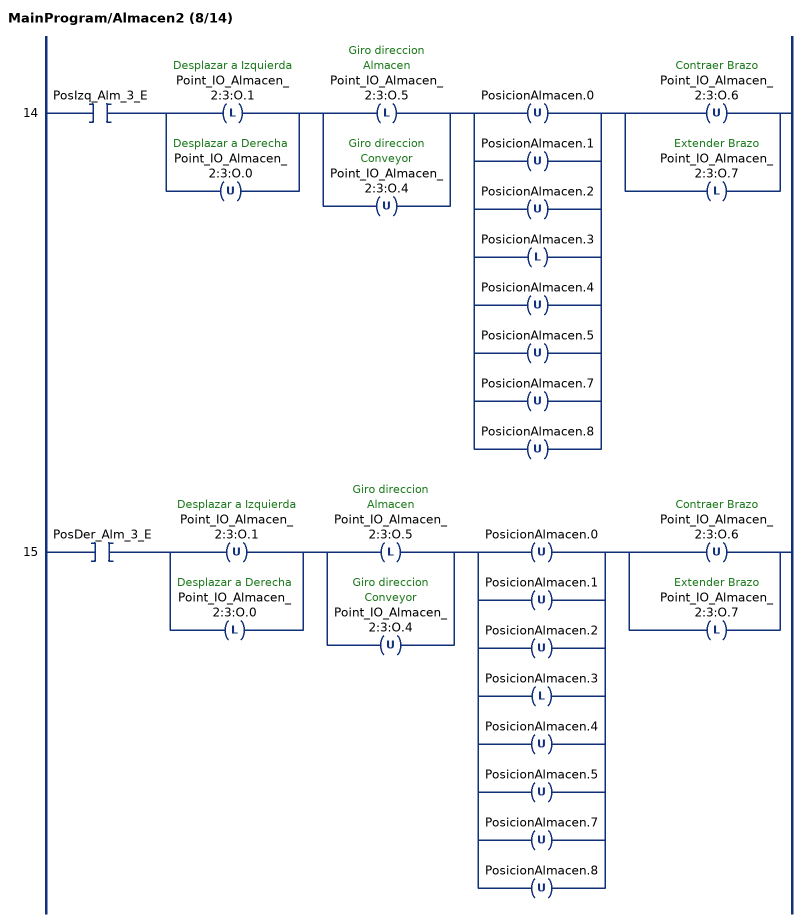
   14: XIC(PosIzq_Alm_3_E)[OTL(Point_IO_Almacen_2:3:O.1) ,OTU(Point_IO_Almacen_2:3:O.0) ][OTL(Point_IO_Almacen_2:3:O.5) ,OTU(Point_IO_Almacen_2:3:O.4) ][OTU(PosicionAlmacen.0) ,OTU(PosicionAlmacen.1) ,OTU(PosicionAlmacen.2) ,OTL(PosicionAlmacen.3) ,OTU(PosicionAlmacen.4) ,OTU(PosicionAlmacen.5) ,OTU(PosicionAlmacen.7) ,OTU(PosicionAlmacen.8) ][OTU(Point_IO_Almacen_2:3:O.6) ,OTL(Point_IO_Almacen_2:3:O.7) ];
   15: XIC(PosDer_Alm_3_E)[OTU(Point_IO_Almacen_2:3:O.1) ,OTL(Point_IO_Almacen_2:3:O.0) ][OTL(Point_IO_Almacen_2:3:O.5) ,OTU(Point_IO_Almacen_2:3:O.4) ][OTU(PosicionAlmacen.0) ,OTU(PosicionAlmacen.1) ,OTU(PosicionAlmacen.2) ,OTL(PosicionAlmacen.3) ,OTU(PosicionAlmacen.4) ,OTU(PosicionAlmacen.5) ,OTU(PosicionAlmacen.7) ,OTU(PosicionAlmacen.8) ][OTU(Point_IO_Almacen_2:3:O.6) ,OTL(Point_IO_Almacen_2:3:O.7) ];
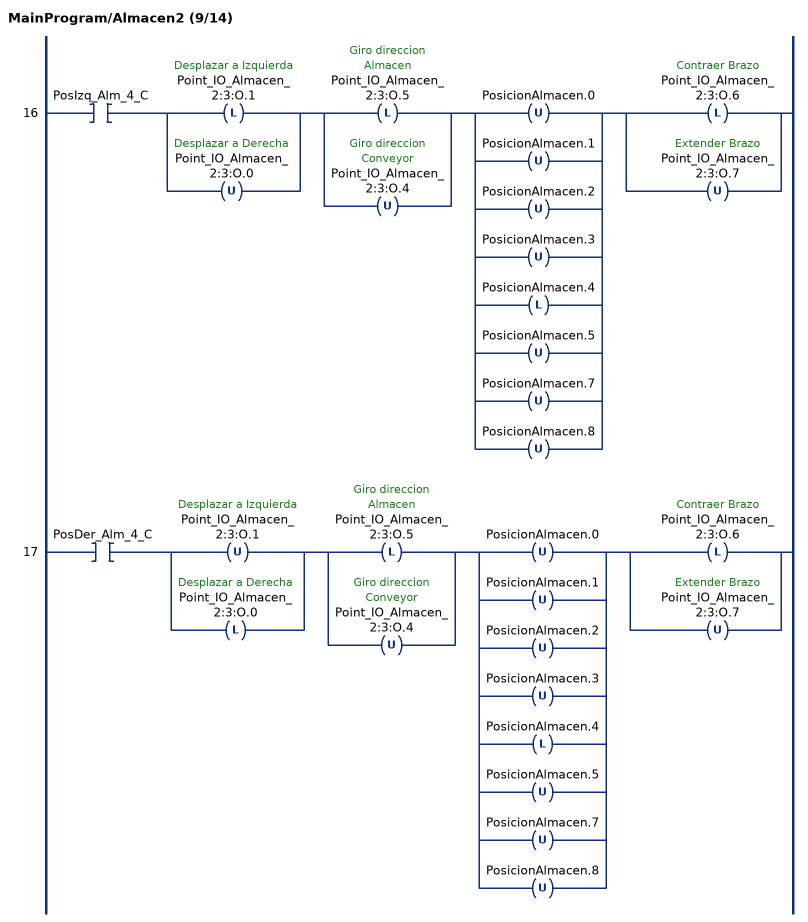
   16: XIC(PosIzq_Alm_4_C)[OTL(Point_IO_Almacen_2:3:O.1) ,OTU(Point_IO_Almacen_2:3:O.0) ][OTL(Point_IO_Almacen_2:3:O.5) ,OTU(Point_IO_Almacen_2:3:O.4) ][OTU(PosicionAlmacen.0) ,OTU(PosicionAlmacen.1) ,OTU(PosicionAlmacen.2) ,OTU(PosicionAlmacen.3) ,OTL(PosicionAlmacen.4) ,OTU(PosicionAlmacen.5) ,OTU(PosicionAlmacen.7) ,OTU(PosicionAlmacen.8) ][OTL(Point_IO_Almacen_2:3:O.6) ,OTU(Point_IO_Almacen_2:3:O.7) ];
   17: XIC(PosDer_Alm_4_C)[OTU(Point_IO_Almacen_2:3:O.1) ,OTL(Point_IO_Almacen_2:3:O.0) ][OTL(Point_IO_Almacen_2:3:O.5) ,OTU(Point_IO_Almacen_2:3:O.4) ][OTU(PosicionAlmacen.0) ,OTU(PosicionAlmacen.1) ,OTU(PosicionAlmacen.2) ,OTU(PosicionAlmacen.3) ,OTL(PosicionAlmacen.4) ,OTU(PosicionAlmacen.5) ,OTU(PosicionAlmacen.7) ,OTU(PosicionAlmacen.8) ][OTL(Point_IO_Almacen_2:3:O.6) ,OTU(Point_IO_Almacen_2:3:O.7) ];
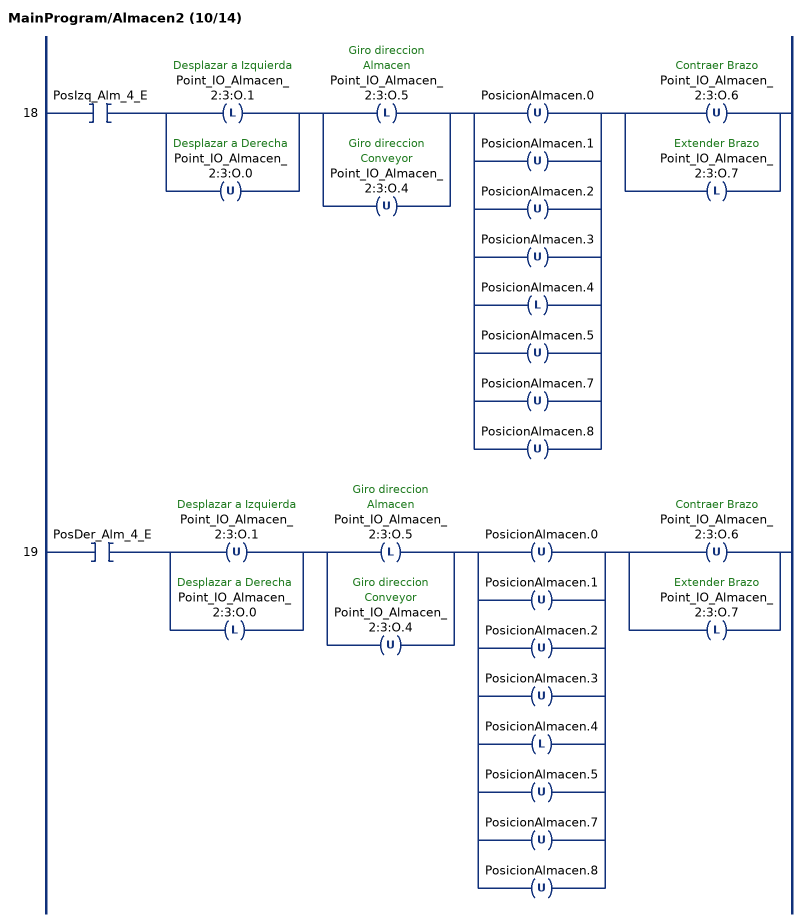
   18: XIC(PosIzq_Alm_4_E)[OTL(Point_IO_Almacen_2:3:O.1) ,OTU(Point_IO_Almacen_2:3:O.0) ][OTL(Point_IO_Almacen_2:3:O.5) ,OTU(Point_IO_Almacen_2:3:O.4) ][OTU(PosicionAlmacen.0) ,OTU(PosicionAlmacen.1) ,OTU(PosicionAlmacen.2) ,OTU(PosicionAlmacen.3) ,OTL(PosicionAlmacen.4) ,OTU(PosicionAlmacen.5) ,OTU(PosicionAlmacen.7) ,OTU(PosicionAlmacen.8) ][OTU(Point_IO_Almacen_2:3:O.6) ,OTL(Point_IO_Almacen_2:3:O.7) ];
   19: XIC(PosDer_Alm_4_E)[OTU(Point_IO_Almacen_2:3:O.1) ,OTL(Point_IO_Almacen_2:3:O.0) ][OTL(Point_IO_Almacen_2:3:O.5) ,OTU(Point_IO_Almacen_2:3:O.4) ][OTU(PosicionAlmacen.0) ,OTU(PosicionAlmacen.1) ,OTU(PosicionAlmacen.2) ,OTU(PosicionAlmacen.3) ,OTL(PosicionAlmacen.4) ,OTU(PosicionAlmacen.5) ,OTU(PosicionAlmacen.7) ,OTU(PosicionAlmacen.8) ][OTU(Point_IO_Almacen_2:3:O.6) ,OTL(Point_IO_Almacen_2:3:O.7) ];
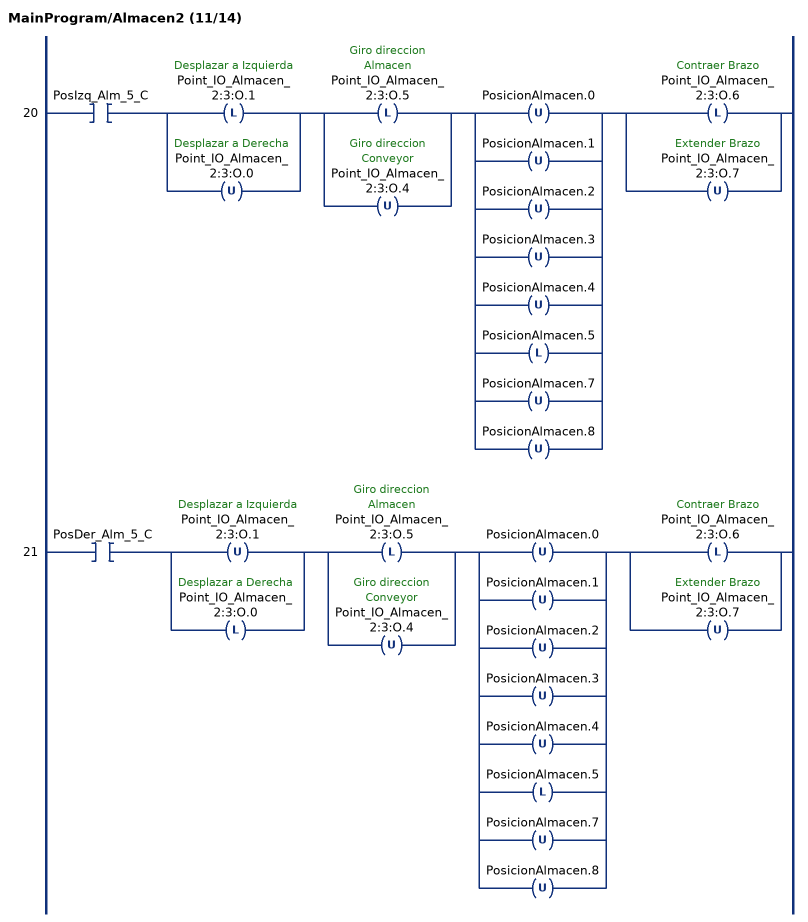
   20: XIC(PosIzq_Alm_5_C)[OTL(Point_IO_Almacen_2:3:O.1) ,OTU(Point_IO_Almacen_2:3:O.0) ][OTL(Point_IO_Almacen_2:3:O.5) ,OTU(Point_IO_Almacen_2:3:O.4) ][OTU(PosicionAlmacen.0) ,OTU(PosicionAlmacen.1) ,OTU(PosicionAlmacen.2) ,OTU(PosicionAlmacen.3) ,OTU(PosicionAlmacen.4) ,OTL(PosicionAlmacen.5) ,OTU(PosicionAlmacen.7) ,OTU(PosicionAlmacen.8) ][OTL(Point_IO_Almacen_2:3:O.6) ,OTU(Point_IO_Almacen_2:3:O.7) ];
   21: XIC(PosDer_Alm_5_C)[OTU(Point_IO_Almacen_2:3:O.1) ,OTL(Point_IO_Almacen_2:3:O.0) ][OTL(Point_IO_Almacen_2:3:O.5) ,OTU(Point_IO_Almacen_2:3:O.4) ][OTU(PosicionAlmacen.0) ,OTU(PosicionAlmacen.1) ,OTU(PosicionAlmacen.2) ,OTU(PosicionAlmacen.3) ,OTU(PosicionAlmacen.4) ,OTL(PosicionAlmacen.5) ,OTU(PosicionAlmacen.7) ,OTU(PosicionAlmacen.8) ][OTL(Point_IO_Almacen_2:3:O.6) ,OTU(Point_IO_Almacen_2:3:O.7) ];
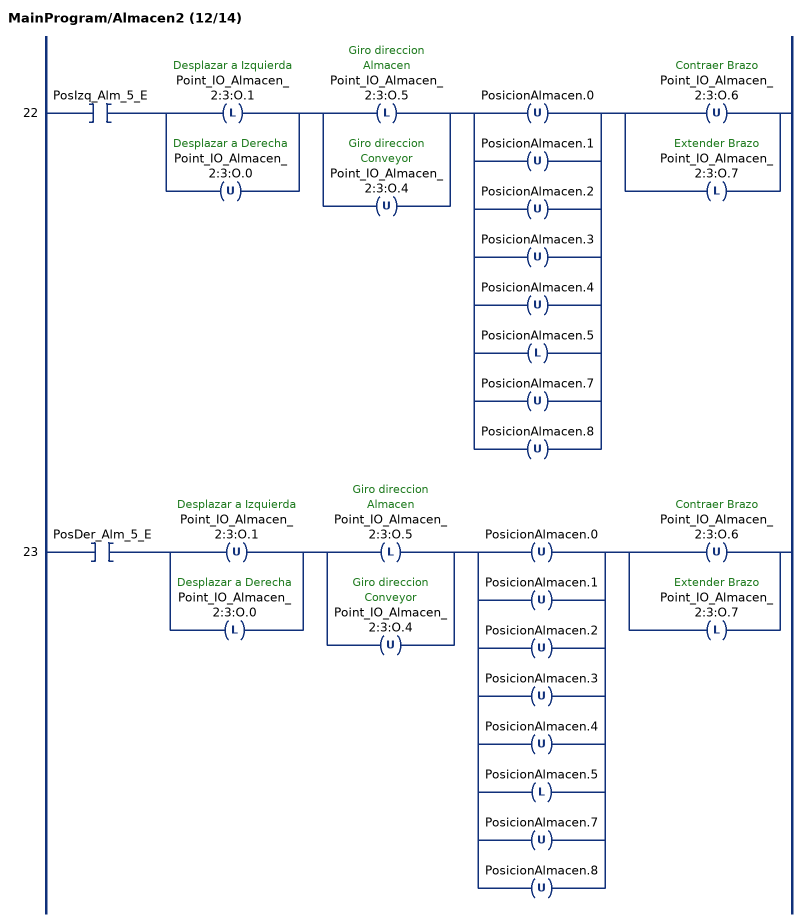
   22: XIC(PosIzq_Alm_5_E)[OTL(Point_IO_Almacen_2:3:O.1) ,OTU(Point_IO_Almacen_2:3:O.0) ][OTL(Point_IO_Almacen_2:3:O.5) ,OTU(Point_IO_Almacen_2:3:O.4) ][OTU(PosicionAlmacen.0) ,OTU(PosicionAlmacen.1) ,OTU(PosicionAlmacen.2) ,OTU(PosicionAlmacen.3) ,OTU(PosicionAlmacen.4) ,OTL(PosicionAlmacen.5) ,OTU(PosicionAlmacen.7) ,OTU(PosicionAlmacen.8) ][OTU(Point_IO_Almacen_2:3:O.6) ,OTL(Point_IO_Almacen_2:3:O.7) ];
   23: XIC(PosDer_Alm_5_E)[OTU(Point_IO_Almacen_2:3:O.1) ,OTL(Point_IO_Almacen_2:3:O.0) ][OTL(Point_IO_Almacen_2:3:O.5) ,OTU(Point_IO_Almacen_2:3:O.4) ][OTU(PosicionAlmacen.0) ,OTU(PosicionAlmacen.1) ,OTU(PosicionAlmacen.2) ,OTU(PosicionAlmacen.3) ,OTU(PosicionAlmacen.4) ,OTL(PosicionAlmacen.5) ,OTU(PosicionAlmacen.7) ,OTU(PosicionAlmacen.8) ][OTU(Point_IO_Almacen_2:3:O.6) ,OTL(Point_IO_Almacen_2:3:O.7) ];
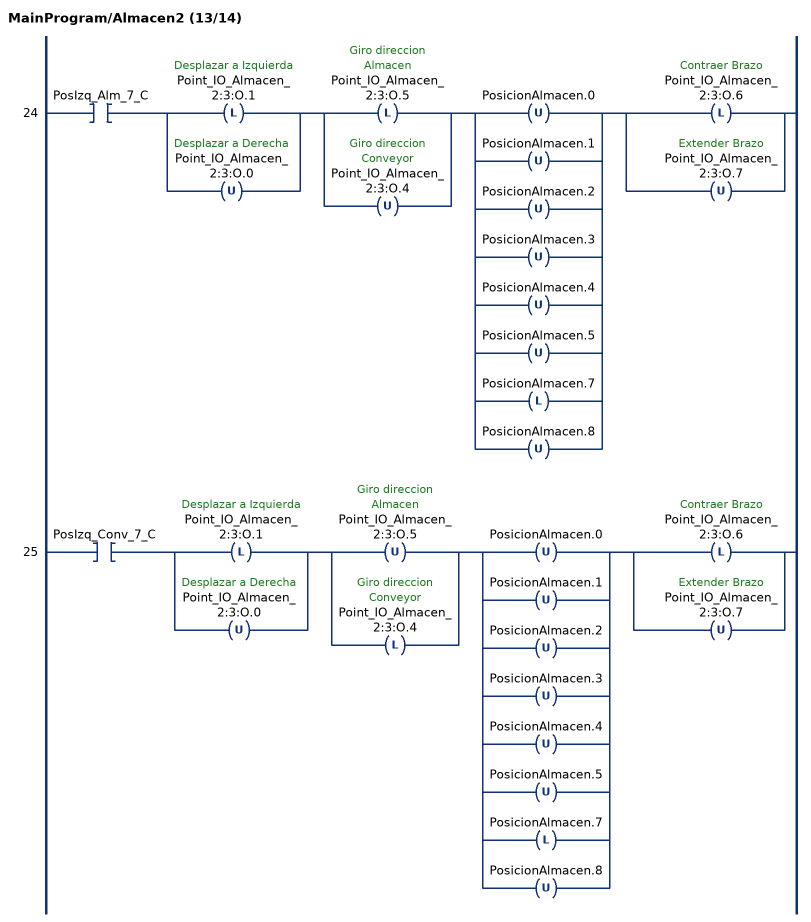
   24: XIC(PosIzq_Alm_7_C)[OTL(Point_IO_Almacen_2:3:O.1) ,OTU(Point_IO_Almacen_2:3:O.0) ][OTL(Point_IO_Almacen_2:3:O.5) ,OTU(Point_IO_Almacen_2:3:O.4) ][OTU(PosicionAlmacen.0) ,OTU(PosicionAlmacen.1) ,OTU(PosicionAlmacen.2) ,OTU(PosicionAlmacen.3) ,OTU(PosicionAlmacen.4) ,OTU(PosicionAlmacen.5) ,OTL(PosicionAlmacen.7) ,OTU(PosicionAlmacen.8) ][OTL(Point_IO_Almacen_2:3:O.6) ,OTU(Point_IO_Almacen_2:3:O.7) ];
   25: XIC(PosIzq_Conv_7_C)[OTL(Point_IO_Almacen_2:3:O.1) ,OTU(Point_IO_Almacen_2:3:O.0) ][OTU(Point_IO_Almacen_2:3:O.5) ,OTL(Point_IO_Almacen_2:3:O.4) ][OTU(PosicionAlmacen.0) ,OTU(PosicionAlmacen.1) ,OTU(PosicionAlmacen.2) ,OTU(PosicionAlmacen.3) ,OTU(PosicionAlmacen.4) ,OTU(PosicionAlmacen.5) ,OTL(PosicionAlmacen.7) ,OTU(PosicionAlmacen.8) ][OTL(Point_IO_Almacen_2:3:O.6) ,OTU(Point_IO_Almacen_2:3:O.7) ];
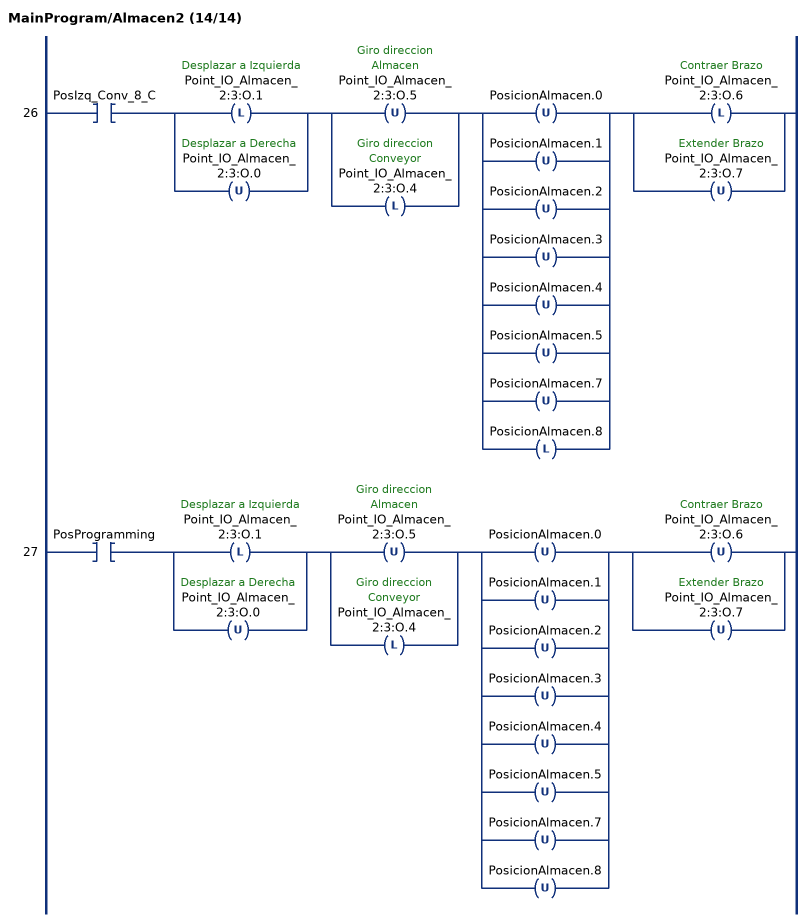
   26: XIC(PosIzq_Conv_8_C)[OTL(Point_IO_Almacen_2:3:O.1) ,OTU(Point_IO_Almacen_2:3:O.0) ][OTU(Point_IO_Almacen_2:3:O.5) ,OTL(Point_IO_Almacen_2:3:O.4) ][OTU(PosicionAlmacen.0) ,OTU(PosicionAlmacen.1) ,OTU(PosicionAlmacen.2) ,OTU(PosicionAlmacen.3) ,OTU(PosicionAlmacen.4) ,OTU(PosicionAlmacen.5) ,OTU(PosicionAlmacen.7) ,OTL(PosicionAlmacen.8) ][OTL(Point_IO_Almacen_2:3:O.6) ,OTU(Point_IO_Almacen_2:3:O.7) ];
   27: XIC(PosProgramming)[OTL(Point_IO_Almacen_2:3:O.1) ,OTU(Point_IO_Almacen_2:3:O.0) ][OTU(Point_IO_Almacen_2:3:O.5) ,OTL(Point_IO_Almacen_2:3:O.4) ][OTU(PosicionAlmacen.0) ,OTU(PosicionAlmacen.1) ,OTU(PosicionAlmacen.2) ,OTU(PosicionAlmacen.3) ,OTU(PosicionAlmacen.4) ,OTU(PosicionAlmacen.5) ,OTU(PosicionAlmacen.7) ,OTU(PosicionAlmacen.8) ][OTU(Point_IO_Almacen_2:3:O.6) ,OTU(Point_IO_Almacen_2:3:O.7) ];
END_ROUTINE
